  [2280] = {x=-3.091, y=2.427, z=22, rx=180, rz=-141.855, shoulder=lefty, elbow=epositive, wrist=wpositive, fatherId=fReference[0]}
  [2281] = {x=-1.854, y=1.456, z=22, rx=-180, rz=-141.854, shoulder=lefty, elbow=epositive, wrist=wpositive, fatherId=fReference[0]}
  [2282] = {x=-0.617, y=0.484, z=22, rx=-180, rz=-141.854, shoulder=lefty, elbow=epositive, wrist=wpositive, fatherId=fReference[0]}
  [2283] = {x=0.62, y=-0.487, z=22, rx=-180, rz=-141.854, shoulder=lefty, elbow=epositive, wrist=wpositive, fatherId=fReference[0]}
  [2284] = {x=1.857, y=-1.459, z=22, rx=180, rz=-141.855, shoulder=lefty, elbow=epositive, wrist=wpositive, fatherId=fReference[0]}
  [2285] = {x=3.094, y=-2.43, z=22, rx=-180, rz=-141.856, shoulder=lefty, elbow=epositive, wrist=wpositive, fatherId=fReference[0]}
  [2286] = {x=4.331, y=-3.402, z=22, rx=180, rz=-141.857, shoulder=lefty, elbow=epositive, wrist=wpositive, fatherId=fReference[0]}
  [2287] = {x=5.568, y=-4.373, z=22, rx=180, rz=-141.859, shoulder=lefty, elbow=epositive, wrist=wpositive, fatherId=fReference[0]}
  [2288] = {x=6.805, y=-5.345, z=22, rx=180, rz=-141.862, shoulder=lefty, elbow=epositive, wrist=wpositive, fatherId=fReference[0]}
  [2289] = {x=8.043, y=-6.316, z=22, rx=-180, rz=-141.864, shoulder=lefty, elbow=epositive, wrist=wpositive, fatherId=fReference[0]}
  [2290] = {x=9.28, y=-7.287, z=22, rx=180, rz=-141.867, shoulder=lefty, elbow=epositive, wrist=wpositive, fatherId=fReference[0]}
  [2291] = {x=10.517, y=-8.259, z=22, rx=-180, rz=-141.871, shoulder=lefty, elbow=epositive, wrist=wpositive, fatherId=fReference[0]}
  [2292] = {x=11.754, y=-9.23, z=22, rx=180, rz=-141.875, shoulder=lefty, elbow=epositive, wrist=wpositive, fatherId=fReference[0]}
  [2293] = {x=12.992, y=-10.201, z=22, rx=-180, rz=-141.879, shoulder=lefty, elbow=epositive, wrist=wpositive, fatherId=fReference[0]}
  [2294] = {x=14.229, y=-11.172, z=22, rx=-180, rz=-141.884, shoulder=lefty, elbow=epositive, wrist=wpositive, fatherId=fReference[0]}
  [2295] = {x=15.467, y=-12.143, z=22, rx=-180, rz=-141.89, shoulder=lefty, elbow=epositive, wrist=wpositive, fatherId=fReference[0]}
  [2296] = {x=16.704, y=-13.113, z=22, rx=180, rz=-141.895, shoulder=lefty, elbow=epositive, wrist=wpositive, fatherId=fReference[0]}
  [2297] = {x=17.942, y=-14.084, z=22, rx=-180, rz=-141.901, shoulder=lefty, elbow=epositive, wrist=wpositive, fatherId=fReference[0]}
  [2298] = {x=19.179, y=-15.054, z=22, rx=-180, rz=-141.908, shoulder=lefty, elbow=epositive, wrist=wpositive, fatherId=fReference[0]}
  [2299] = {x=20.417, y=-16.025, z=22, rx=-180, rz=-141.915, shoulder=lefty, elbow=epositive, wrist=wpositive, fatherId=fReference[0]}
  [2300] = {x=21.655, y=-16.995, z=22, rx=-180, rz=-141.922, shoulder=lefty, elbow=epositive, wrist=wpositive, fatherId=fReference[0]}
  [2301] = {x=22.893, y=-17.965, z=22, rx=180, rz=-141.93, shoulder=lefty, elbow=epositive, wrist=wpositive, fatherId=fReference[0]}
  [2302] = {x=24.131, y=-18.934, z=22, rx=-180, rz=-141.938, shoulder=lefty, elbow=epositive, wrist=wpositive, fatherId=fReference[0]}
  [2303] = {x=25.369, y=-19.904, z=22, rx=-180, rz=-141.947, shoulder=lefty, elbow=epositive, wrist=wpositive, fatherId=fReference[0]}
  [2304] = {x=26.607, y=-20.873, z=22, rx=180, rz=-141.956, shoulder=lefty, elbow=epositive, wrist=wpositive, fatherId=fReference[0]}
  [2305] = {x=27.846, y=-21.842, z=22, rx=180, rz=-141.965, shoulder=lefty, elbow=epositive, wrist=wpositive, fatherId=fReference[0]}
  [2306] = {x=29.084, y=-22.811, z=22, rx=180, rz=-141.975, shoulder=lefty, elbow=epositive, wrist=wpositive, fatherId=fReference[0]}
  [2307] = {x=30.323, y=-23.779, z=22, rx=-180, rz=-141.986, shoulder=lefty, elbow=epositive, wrist=wpositive, fatherId=fReference[0]}
  [2308] = {x=31.561, y=-24.748, z=22, rx=-180, rz=-141.996, shoulder=lefty, elbow=epositive, wrist=wpositive, fatherId=fReference[0]}
  [2309] = {x=32.8, y=-25.716, z=22, rx=180, rz=-142.008, shoulder=lefty, elbow=epositive, wrist=wpositive, fatherId=fReference[0]}
  [2310] = {x=34.039, y=-26.683, z=22, rx=-180, rz=-142.019, shoulder=lefty, elbow=epositive, wrist=wpositive, fatherId=fReference[0]}
  [2311] = {x=35.278, y=-27.651, z=22, rx=-180, rz=-142.031, shoulder=lefty, elbow=epositive, wrist=wpositive, fatherId=fReference[0]}
  [2312] = {x=36.517, y=-28.618, z=22, rx=-180, rz=-142.044, shoulder=lefty, elbow=epositive, wrist=wpositive, fatherId=fReference[0]}
  [2313] = {x=37.757, y=-29.585, z=22, rx=180, rz=-142.057, shoulder=lefty, elbow=epositive, wrist=wpositive, fatherId=fReference[0]}
  [2314] = {x=38.996, y=-30.551, z=22, rx=-180, rz=-142.07, shoulder=lefty, elbow=epositive, wrist=wpositive, fatherId=fReference[0]}
  [2315] = {x=40.236, y=-31.517, z=22, rx=180, rz=-142.084, shoulder=lefty, elbow=epositive, wrist=wpositive, fatherId=fReference[0]}
  [2316] = {x=41.476, y=-32.483, z=22, rx=180, rz=-142.098, shoulder=lefty, elbow=epositive, wrist=wpositive, fatherId=fReference[0]}
  [2317] = {x=42.715, y=-33.448, z=22, rx=-180, rz=-142.113, shoulder=lefty, elbow=epositive, wrist=wpositive, fatherId=fReference[0]}
  [2318] = {x=43.956, y=-34.413, z=22, rx=180, rz=-142.128, shoulder=lefty, elbow=epositive, wrist=wpositive, fatherId=fReference[0]}
  [2319] = {x=45.196, y=-35.377, z=22, rx=180, rz=-142.143, shoulder=lefty, elbow=epositive, wrist=wpositive, fatherId=fReference[0]}
  [2320] = {x=46.436, y=-36.342, z=22, rx=180, rz=-142.159, shoulder=lefty, elbow=epositive, wrist=wpositive, fatherId=fReference[0]}
  [2321] = {x=47.677, y=-37.305, z=22, rx=-180, rz=-142.175, shoulder=lefty, elbow=epositive, wrist=wpositive, fatherId=fReference[0]}
  [2322] = {x=48.917, y=-38.269, z=22, rx=-180, rz=-142.192, shoulder=lefty, elbow=epositive, wrist=wpositive, fatherId=fReference[0]}
  [2323] = {x=50.158, y=-39.231, z=22, rx=180, rz=-142.209, shoulder=lefty, elbow=epositive, wrist=wpositive, fatherId=fReference[0]}
  [2324] = {x=51.399, y=-40.194, z=22, rx=-180, rz=-142.227, shoulder=lefty, elbow=epositive, wrist=wpositive, fatherId=fReference[0]}
  [2325] = {x=52.641, y=-41.156, z=22, rx=180, rz=-142.245, shoulder=lefty, elbow=epositive, wrist=wpositive, fatherId=fReference[0]}
  [2326] = {x=53.882, y=-42.117, z=22, rx=-180, rz=-142.263, shoulder=lefty, elbow=epositive, wrist=wpositive, fatherId=fReference[0]}
  [2327] = {x=55.124, y=-43.078, z=22, rx=-180, rz=-142.282, shoulder=lefty, elbow=epositive, wrist=wpositive, fatherId=fReference[0]}
  [2328] = {x=56.366, y=-44.038, z=22, rx=180, rz=-142.302, shoulder=lefty, elbow=epositive, wrist=wpositive, fatherId=fReference[0]}
  [2329] = {x=57.608, y=-44.998, z=22, rx=-180, rz=-142.321, shoulder=lefty, elbow=epositive, wrist=wpositive, fatherId=fReference[0]}
  [2330] = {x=58.85, y=-45.958, z=22, rx=-180, rz=-142.342, shoulder=lefty, elbow=epositive, wrist=wpositive, fatherId=fReference[0]}
  [2331] = {x=60.092, y=-46.916, z=22, rx=-180, rz=-142.362, shoulder=lefty, elbow=epositive, wrist=wpositive, fatherId=fReference[0]}
  [2332] = {x=61.335, y=-47.875, z=22, rx=180, rz=-142.383, shoulder=lefty, elbow=epositive, wrist=wpositive, fatherId=fReference[0]}
  [2333] = {x=62.578, y=-48.832, z=22, rx=-180, rz=-142.405, shoulder=lefty, elbow=epositive, wrist=wpositive, fatherId=fReference[0]}
  [2334] = {x=63.821, y=-49.79, z=22, rx=-180, rz=-142.427, shoulder=lefty, elbow=epositive, wrist=wpositive, fatherId=fReference[0]}
  [2335] = {x=65.064, y=-50.746, z=22, rx=-180, rz=-142.449, shoulder=lefty, elbow=epositive, wrist=wpositive, fatherId=fReference[0]}
  [2336] = {x=66.308, y=-51.702, z=22, rx=-180, rz=-142.472, shoulder=lefty, elbow=epositive, wrist=wpositive, fatherId=fReference[0]}
  [2337] = {x=67.551, y=-52.657, z=22, rx=180, rz=-142.496, shoulder=lefty, elbow=epositive, wrist=wpositive, fatherId=fReference[0]}
  [2338] = {x=68.795, y=-53.612, z=22, rx=180, rz=-142.519, shoulder=lefty, elbow=epositive, wrist=wpositive, fatherId=fReference[0]}
  [2339] = {x=70.04, y=-54.566, z=22, rx=-180, rz=-142.543, shoulder=lefty, elbow=epositive, wrist=wpositive, fatherId=fReference[0]}
  [2340] = {x=71.284, y=-55.519, z=22, rx=-180, rz=-142.568, shoulder=lefty, elbow=epositive, wrist=wpositive, fatherId=fReference[0]}
  [2341] = {x=72.529, y=-56.472, z=22, rx=180, rz=-142.593, shoulder=lefty, elbow=epositive, wrist=wpositive, fatherId=fReference[0]}
  [2342] = {x=73.774, y=-57.424, z=22, rx=-180, rz=-142.619, shoulder=lefty, elbow=epositive, wrist=wpositive, fatherId=fReference[0]}
  [2343] = {x=75.019, y=-58.376, z=22, rx=180, rz=-142.645, shoulder=lefty, elbow=epositive, wrist=wpositive, fatherId=fReference[0]}
  [2344] = {x=76.264, y=-59.326, z=22, rx=-180, rz=-142.671, shoulder=lefty, elbow=epositive, wrist=wpositive, fatherId=fReference[0]}
  [2345] = {x=77.51, y=-60.276, z=22, rx=-180, rz=-142.698, shoulder=lefty, elbow=epositive, wrist=wpositive, fatherId=fReference[0]}
  [2346] = {x=78.756, y=-61.226, z=22, rx=-180, rz=-142.725, shoulder=lefty, elbow=epositive, wrist=wpositive, fatherId=fReference[0]}
  [2347] = {x=80.002, y=-62.174, z=22, rx=180, rz=-142.753, shoulder=lefty, elbow=epositive, wrist=wpositive, fatherId=fReference[0]}
  [2348] = {x=81.249, y=-63.122, z=22, rx=180, rz=-142.781, shoulder=lefty, elbow=epositive, wrist=wpositive, fatherId=fReference[0]}
  [2349] = {x=82.496, y=-64.069, z=22, rx=180, rz=-142.81, shoulder=lefty, elbow=epositive, wrist=wpositive, fatherId=fReference[0]}
  [2350] = {x=83.743, y=-65.015, z=22, rx=180, rz=-142.839, shoulder=lefty, elbow=epositive, wrist=wpositive, fatherId=fReference[0]}
  [2351] = {x=84.99, y=-65.961, z=22, rx=-180, rz=-142.868, shoulder=lefty, elbow=epositive, wrist=wpositive, fatherId=fReference[0]}
  [2352] = {x=86.238, y=-66.905, z=22, rx=-180, rz=-142.898, shoulder=lefty, elbow=epositive, wrist=wpositive, fatherId=fReference[0]}
  [2353] = {x=87.486, y=-67.849, z=22, rx=-180, rz=-142.929, shoulder=lefty, elbow=epositive, wrist=wpositive, fatherId=fReference[0]}
  [2354] = {x=88.734, y=-68.792, z=22, rx=-180, rz=-142.96, shoulder=lefty, elbow=epositive, wrist=wpositive, fatherId=fReference[0]}
  [2355] = {x=89.982, y=-69.734, z=22, rx=-180, rz=-142.991, shoulder=lefty, elbow=epositive, wrist=wpositive, fatherId=fReference[0]}
  [2356] = {x=91.231, y=-70.676, z=22, rx=-180, rz=-143.023, shoulder=lefty, elbow=epositive, wrist=wpositive, fatherId=fReference[0]}
  [2357] = {x=92.48, y=-71.616, z=22, rx=180, rz=-143.055, shoulder=lefty, elbow=epositive, wrist=wpositive, fatherId=fReference[0]}
  [2358] = {x=93.73, y=-72.556, z=22, rx=-180, rz=-143.088, shoulder=lefty, elbow=epositive, wrist=wpositive, fatherId=fReference[0]}
  [2359] = {x=94.979, y=-73.495, z=22, rx=-180, rz=-143.121, shoulder=lefty, elbow=epositive, wrist=wpositive, fatherId=fReference[0]}
  [2360] = {x=96.23, y=-74.432, z=22, rx=-180, rz=-143.155, shoulder=lefty, elbow=epositive, wrist=wpositive, fatherId=fReference[0]}
  [2361] = {x=97.48, y=-75.369, z=22, rx=180, rz=-143.189, shoulder=lefty, elbow=epositive, wrist=wpositive, fatherId=fReference[0]}
  [2362] = {x=98.731, y=-76.305, z=22, rx=-180, rz=-143.224, shoulder=lefty, elbow=epositive, wrist=wpositive, fatherId=fReference[0]}
  [2363] = {x=99.982, y=-77.24, z=22, rx=-180, rz=-143.259, shoulder=lefty, elbow=epositive, wrist=wpositive, fatherId=fReference[0]}
  [2364] = {x=101.233, y=-78.175, z=22, rx=-180, rz=-143.294, shoulder=lefty, elbow=epositive, wrist=wpositive, fatherId=fReference[0]}
  [2365] = {x=102.485, y=-79.108, z=22, rx=180, rz=-143.33, shoulder=lefty, elbow=epositive, wrist=wpositive, fatherId=fReference[0]}
  [2366] = {x=103.737, y=-80.04, z=22, rx=-180, rz=-143.367, shoulder=lefty, elbow=epositive, wrist=wpositive, fatherId=fReference[0]}
  [2367] = {x=104.989, y=-80.971, z=22, rx=-180, rz=-143.404, shoulder=lefty, elbow=epositive, wrist=wpositive, fatherId=fReference[0]}
  [2368] = {x=106.242, y=-81.901, z=22, rx=-180, rz=-143.441, shoulder=lefty, elbow=epositive, wrist=wpositive, fatherId=fReference[0]}
  [2369] = {x=107.495, y=-82.831, z=22, rx=-180, rz=-143.479, shoulder=lefty, elbow=epositive, wrist=wpositive, fatherId=fReference[0]}
  [2370] = {x=108.748, y=-83.759, z=22, rx=180, rz=-143.517, shoulder=lefty, elbow=epositive, wrist=wpositive, fatherId=fReference[0]}
  [2371] = {x=110.002, y=-84.686, z=22, rx=-180, rz=-143.556, shoulder=lefty, elbow=epositive, wrist=wpositive, fatherId=fReference[0]}
  [2372] = {x=111.256, y=-85.612, z=22, rx=-180, rz=-143.596, shoulder=lefty, elbow=epositive, wrist=wpositive, fatherId=fReference[0]}
  [2373] = {x=112.511, y=-86.537, z=22, rx=-180, rz=-143.635, shoulder=lefty, elbow=epositive, wrist=wpositive, fatherId=fReference[0]}
  [2374] = {x=113.766, y=-87.461, z=22, rx=180, rz=-143.676, shoulder=lefty, elbow=epositive, wrist=wpositive, fatherId=fReference[0]}
  [2375] = {x=115.021, y=-88.384, z=22, rx=180, rz=-143.716, shoulder=lefty, elbow=epositive, wrist=wpositive, fatherId=fReference[0]}
  [2376] = {x=116.277, y=-89.306, z=22, rx=-180, rz=-143.758, shoulder=lefty, elbow=epositive, wrist=wpositive, fatherId=fReference[0]}
  [2377] = {x=117.533, y=-90.227, z=22, rx=-180, rz=-143.799, shoulder=lefty, elbow=epositive, wrist=wpositive, fatherId=fReference[0]}
  [2378] = {x=118.789, y=-91.146, z=22, rx=-180, rz=-143.842, shoulder=lefty, elbow=epositive, wrist=wpositive, fatherId=fReference[0]}
  [2379] = {x=120.046, y=-92.065, z=22, rx=-180, rz=-143.884, shoulder=lefty, elbow=epositive, wrist=wpositive, fatherId=fReference[0]}
  [2380] = {x=121.304, y=-92.982, z=22, rx=-180, rz=-143.927, shoulder=lefty, elbow=epositive, wrist=wpositive, fatherId=fReference[0]}
  [2381] = {x=122.561, y=-93.898, z=22, rx=180, rz=-143.971, shoulder=lefty, elbow=epositive, wrist=wpositive, fatherId=fReference[0]}
  [2382] = {x=123.819, y=-94.813, z=22, rx=-180, rz=-144.015, shoulder=lefty, elbow=epositive, wrist=wpositive, fatherId=fReference[0]}
  [2383] = {x=125.078, y=-95.727, z=22, rx=180, rz=-144.06, shoulder=lefty, elbow=epositive, wrist=wpositive, fatherId=fReference[0]}
  [2384] = {x=126.337, y=-96.64, z=22, rx=-180, rz=-144.105, shoulder=lefty, elbow=epositive, wrist=wpositive, fatherId=fReference[0]}
  [2385] = {x=127.596, y=-97.551, z=22, rx=-180, rz=-144.151, shoulder=lefty, elbow=epositive, wrist=wpositive, fatherId=fReference[0]}
  [2386] = {x=128.856, y=-98.461, z=22, rx=-180, rz=-144.197, shoulder=lefty, elbow=epositive, wrist=wpositive, fatherId=fReference[0]}
  [2387] = {x=130.116, y=-99.37, z=22, rx=180, rz=-144.243, shoulder=lefty, elbow=epositive, wrist=wpositive, fatherId=fReference[0]}
  [2388] = {x=131.376, y=-100.278, z=22, rx=-180, rz=-144.291, shoulder=lefty, elbow=epositive, wrist=wpositive, fatherId=fReference[0]}
  [2389] = {x=132.637, y=-101.185, z=22, rx=180, rz=-144.338, shoulder=lefty, elbow=epositive, wrist=wpositive, fatherId=fReference[0]}
  [2390] = {x=133.899, y=-102.09, z=22, rx=-180, rz=-144.386, shoulder=lefty, elbow=epositive, wrist=wpositive, fatherId=fReference[0]}
  [2391] = {x=135.161, y=-102.994, z=22, rx=-180, rz=-144.435, shoulder=lefty, elbow=epositive, wrist=wpositive, fatherId=fReference[0]}
  [2392] = {x=136.423, y=-103.896, z=22, rx=180, rz=-144.484, shoulder=lefty, elbow=epositive, wrist=wpositive, fatherId=fReference[0]}
  [2393] = {x=137.686, y=-104.798, z=22, rx=180, rz=-144.534, shoulder=lefty, elbow=epositive, wrist=wpositive, fatherId=fReference[0]}
  [2394] = {x=138.949, y=-105.698, z=22, rx=180, rz=-144.584, shoulder=lefty, elbow=epositive, wrist=wpositive, fatherId=fReference[0]}
  [2395] = {x=140.213, y=-106.596, z=22, rx=180, rz=-144.634, shoulder=lefty, elbow=epositive, wrist=wpositive, fatherId=fReference[0]}
  [2396] = {x=141.477, y=-107.494, z=22, rx=-180, rz=-144.686, shoulder=lefty, elbow=epositive, wrist=wpositive, fatherId=fReference[0]}
  [2397] = {x=142.742, y=-108.389, z=22, rx=-180, rz=-144.737, shoulder=lefty, elbow=epositive, wrist=wpositive, fatherId=fReference[0]}
  [2398] = {x=144.007, y=-109.284, z=22, rx=-180, rz=-144.789, shoulder=lefty, elbow=epositive, wrist=wpositive, fatherId=fReference[0]}
  [2399] = {x=145.273, y=-110.177, z=22, rx=-180, rz=-144.842, shoulder=lefty, elbow=epositive, wrist=wpositive, fatherId=fReference[0]}
  [2400] = {x=146.539, y=-111.069, z=22, rx=-180, rz=-144.895, shoulder=lefty, elbow=epositive, wrist=wpositive, fatherId=fReference[0]}
  [2401] = {x=147.806, y=-111.959, z=22, rx=-180, rz=-144.949, shoulder=lefty, elbow=epositive, wrist=wpositive, fatherId=fReference[0]}
  [2402] = {x=149.073, y=-112.848, z=22, rx=-180, rz=-145.003, shoulder=lefty, elbow=epositive, wrist=wpositive, fatherId=fReference[0]}
  [2403] = {x=150.34, y=-113.736, z=22, rx=-180, rz=-145.058, shoulder=lefty, elbow=epositive, wrist=wpositive, fatherId=fReference[0]}
  [2404] = {x=151.608, y=-114.622, z=22, rx=-180, rz=-145.113, shoulder=lefty, elbow=epositive, wrist=wpositive, fatherId=fReference[0]}
  [2405] = {x=152.877, y=-115.506, z=22, rx=-180, rz=-145.169, shoulder=lefty, elbow=epositive, wrist=wpositive, fatherId=fReference[0]}
  [2406] = {x=154.146, y=-116.389, z=22, rx=180, rz=-145.225, shoulder=lefty, elbow=epositive, wrist=wpositive, fatherId=fReference[0]}
  [2407] = {x=155.416, y=-117.271, z=22, rx=180, rz=-145.282, shoulder=lefty, elbow=epositive, wrist=wpositive, fatherId=fReference[0]}
  [2408] = {x=156.686, y=-118.151, z=22, rx=-180, rz=-145.34, shoulder=lefty, elbow=epositive, wrist=wpositive, fatherId=fReference[0]}
  [2409] = {x=157.957, y=-119.03, z=22, rx=180, rz=-145.398, shoulder=lefty, elbow=epositive, wrist=wpositive, fatherId=fReference[0]}
  [2410] = {x=159.228, y=-119.907, z=22, rx=-180, rz=-145.456, shoulder=lefty, elbow=epositive, wrist=wpositive, fatherId=fReference[0]}
  [2411] = {x=160.5, y=-120.782, z=22, rx=-180, rz=-145.515, shoulder=lefty, elbow=epositive, wrist=wpositive, fatherId=fReference[0]}
  [2412] = {x=161.772, y=-121.656, z=22, rx=180, rz=-145.575, shoulder=lefty, elbow=epositive, wrist=wpositive, fatherId=fReference[0]}
  [2413] = {x=163.045, y=-122.529, z=22, rx=-180, rz=-145.635, shoulder=lefty, elbow=epositive, wrist=wpositive, fatherId=fReference[0]}
  [2414] = {x=164.319, y=-123.4, z=22, rx=-180, rz=-145.695, shoulder=lefty, elbow=epositive, wrist=wpositive, fatherId=fReference[0]}
  [2415] = {x=165.593, y=-124.269, z=22, rx=-180, rz=-145.756, shoulder=lefty, elbow=epositive, wrist=wpositive, fatherId=fReference[0]}
  [2416] = {x=166.867, y=-125.136, z=22, rx=-180, rz=-145.818, shoulder=lefty, elbow=epositive, wrist=wpositive, fatherId=fReference[0]}
  [2417] = {x=168.142, y=-126.002, z=22, rx=-180, rz=-145.88, shoulder=lefty, elbow=epositive, wrist=wpositive, fatherId=fReference[0]}
  [2418] = {x=169.418, y=-126.867, z=22, rx=-180, rz=-145.943, shoulder=lefty, elbow=epositive, wrist=wpositive, fatherId=fReference[0]}
  [2419] = {x=170.695, y=-127.73, z=22, rx=180, rz=-146.006, shoulder=lefty, elbow=epositive, wrist=wpositive, fatherId=fReference[0]}
  [2420] = {x=171.971, y=-128.591, z=22, rx=180, rz=-146.07, shoulder=lefty, elbow=epositive, wrist=wpositive, fatherId=fReference[0]}
  [2421] = {x=173.249, y=-129.45, z=22, rx=-180, rz=-146.135, shoulder=lefty, elbow=epositive, wrist=wpositive, fatherId=fReference[0]}
  [2422] = {x=174.527, y=-130.308, z=22, rx=180, rz=-146.2, shoulder=lefty, elbow=epositive, wrist=wpositive, fatherId=fReference[0]}
  [2423] = {x=175.806, y=-131.164, z=22, rx=-180, rz=-146.265, shoulder=lefty, elbow=epositive, wrist=wpositive, fatherId=fReference[0]}
  [2424] = {x=177.085, y=-132.018, z=22, rx=180, rz=-146.331, shoulder=lefty, elbow=epositive, wrist=wpositive, fatherId=fReference[0]}
  [2425] = {x=178.365, y=-132.871, z=22, rx=-180, rz=-146.398, shoulder=lefty, elbow=epositive, wrist=wpositive, fatherId=fReference[0]}
  [2426] = {x=179.645, y=-133.721, z=22, rx=-180, rz=-146.465, shoulder=lefty, elbow=epositive, wrist=wpositive, fatherId=fReference[0]}
  [2427] = {x=180.927, y=-134.571, z=22, rx=180, rz=-146.533, shoulder=lefty, elbow=epositive, wrist=wpositive, fatherId=fReference[0]}
  [2428] = {x=182.208, y=-135.418, z=22, rx=-180, rz=-146.601, shoulder=lefty, elbow=epositive, wrist=wpositive, fatherId=fReference[0]}
  [2429] = {x=183.491, y=-136.263, z=22, rx=-180, rz=-146.67, shoulder=lefty, elbow=epositive, wrist=wpositive, fatherId=fReference[0]}
  [2430] = {x=184.774, y=-137.107, z=22, rx=180, rz=-146.74, shoulder=lefty, elbow=epositive, wrist=wpositive, fatherId=fReference[0]}
  [2431] = {x=186.057, y=-137.949, z=22, rx=-180, rz=-146.81, shoulder=lefty, elbow=epositive, wrist=wpositive, fatherId=fReference[0]}
  [2432] = {x=187.341, y=-138.789, z=22, rx=180, rz=-146.881, shoulder=lefty, elbow=epositive, wrist=wpositive, fatherId=fReference[0]}
  [2433] = {x=188.626, y=-139.627, z=22, rx=-180, rz=-146.952, shoulder=lefty, elbow=epositive, wrist=wpositive, fatherId=fReference[0]}
  [2434] = {x=189.912, y=-140.464, z=22, rx=-180, rz=-147.024, shoulder=lefty, elbow=epositive, wrist=wpositive, fatherId=fReference[0]}
  [2435] = {x=191.198, y=-141.298, z=22, rx=-180, rz=-147.096, shoulder=lefty, elbow=epositive, wrist=wpositive, fatherId=fReference[0]}
  [2436] = {x=192.485, y=-142.131, z=22, rx=-180, rz=-147.169, shoulder=lefty, elbow=epositive, wrist=wpositive, fatherId=fReference[0]}
  [2437] = {x=193.772, y=-142.961, z=22, rx=-180, rz=-147.243, shoulder=lefty, elbow=epositive, wrist=wpositive, fatherId=fReference[0]}
  [2438] = {x=195.06, y=-143.79, z=22, rx=-180, rz=-147.317, shoulder=lefty, elbow=epositive, wrist=wpositive, fatherId=fReference[0]}
  [2439] = {x=196.349, y=-144.617, z=22, rx=-180, rz=-147.392, shoulder=lefty, elbow=epositive, wrist=wpositive, fatherId=fReference[0]}
  [2440] = {x=197.639, y=-145.442, z=22, rx=-180, rz=-147.467, shoulder=lefty, elbow=epositive, wrist=wpositive, fatherId=fReference[0]}
  [2441] = {x=198.929, y=-146.265, z=22, rx=-180, rz=-147.543, shoulder=lefty, elbow=epositive, wrist=wpositive, fatherId=fReference[0]}
  [2442] = {x=200.219, y=-147.086, z=22, rx=180, rz=-147.619, shoulder=lefty, elbow=epositive, wrist=wpositive, fatherId=fReference[0]}
  [2443] = {x=201.511, y=-147.905, z=22, rx=-180, rz=-147.697, shoulder=lefty, elbow=epositive, wrist=wpositive, fatherId=fReference[0]}
  [2444] = {x=202.803, y=-148.722, z=22, rx=-180, rz=-147.774, shoulder=lefty, elbow=epositive, wrist=wpositive, fatherId=fReference[0]}
  [2445] = {x=204.096, y=-149.536, z=22, rx=-180, rz=-147.853, shoulder=lefty, elbow=epositive, wrist=wpositive, fatherId=fReference[0]}
  [2446] = {x=205.389, y=-150.349, z=22, rx=-180, rz=-147.931, shoulder=lefty, elbow=epositive, wrist=wpositive, fatherId=fReference[0]}
  [2447] = {x=206.683, y=-151.16, z=22, rx=180, rz=-148.011, shoulder=lefty, elbow=epositive, wrist=wpositive, fatherId=fReference[0]}
  [2448] = {x=207.978, y=-151.969, z=22, rx=-180, rz=-148.091, shoulder=lefty, elbow=epositive, wrist=wpositive, fatherId=fReference[0]}
  [2449] = {x=209.273, y=-152.775, z=22, rx=-180, rz=-148.172, shoulder=lefty, elbow=epositive, wrist=wpositive, fatherId=fReference[0]}
  [2450] = {x=210.569, y=-153.58, z=22, rx=-180, rz=-148.253, shoulder=lefty, elbow=epositive, wrist=wpositive, fatherId=fReference[0]}
  [2451] = {x=211.866, y=-154.382, z=22, rx=-180, rz=-148.335, shoulder=lefty, elbow=epositive, wrist=wpositive, fatherId=fReference[0]}
  [2452] = {x=213.164, y=-155.183, z=22, rx=-180, rz=-148.418, shoulder=lefty, elbow=epositive, wrist=wpositive, fatherId=fReference[0]}
  [2453] = {x=214.462, y=-155.981, z=22, rx=-180, rz=-148.501, shoulder=lefty, elbow=epositive, wrist=wpositive, fatherId=fReference[0]}
  [2454] = {x=215.761, y=-156.777, z=22, rx=180, rz=-148.585, shoulder=lefty, elbow=epositive, wrist=wpositive, fatherId=fReference[0]}
  [2455] = {x=217.06, y=-157.57, z=22, rx=-180, rz=-148.669, shoulder=lefty, elbow=epositive, wrist=wpositive, fatherId=fReference[0]}
  [2456] = {x=218.361, y=-158.362, z=22, rx=-180, rz=-148.754, shoulder=lefty, elbow=epositive, wrist=wpositive, fatherId=fReference[0]}
  [2457] = {x=219.662, y=-159.151, z=22, rx=-180, rz=-148.84, shoulder=lefty, elbow=epositive, wrist=wpositive, fatherId=fReference[0]}
  [2458] = {x=220.963, y=-159.938, z=22, rx=-180, rz=-148.926, shoulder=lefty, elbow=epositive, wrist=wpositive, fatherId=fReference[0]}
  [2459] = {x=222.266, y=-160.723, z=22, rx=-180, rz=-149.013, shoulder=lefty, elbow=epositive, wrist=wpositive, fatherId=fReference[0]}
  [2460] = {x=223.569, y=-161.506, z=22, rx=-180, rz=-149.101, shoulder=lefty, elbow=epositive, wrist=wpositive, fatherId=fReference[0]}
  [2461] = {x=224.872, y=-162.286, z=22, rx=180, rz=-149.189, shoulder=lefty, elbow=epositive, wrist=wpositive, fatherId=fReference[0]}
  [2462] = {x=226.177, y=-163.064, z=22, rx=180, rz=-149.278, shoulder=lefty, elbow=epositive, wrist=wpositive, fatherId=fReference[0]}
  [2463] = {x=227.482, y=-163.84, z=22, rx=-180, rz=-149.367, shoulder=lefty, elbow=epositive, wrist=wpositive, fatherId=fReference[0]}
  [2464] = {x=228.788, y=-164.613, z=22, rx=-180, rz=-149.458, shoulder=lefty, elbow=epositive, wrist=wpositive, fatherId=fReference[0]}
  [2465] = {x=230.095, y=-165.384, z=22, rx=180, rz=-149.548, shoulder=lefty, elbow=epositive, wrist=wpositive, fatherId=fReference[0]}
  [2466] = {x=231.402, y=-166.152, z=22, rx=-180, rz=-149.64, shoulder=lefty, elbow=epositive, wrist=wpositive, fatherId=fReference[0]}
  [2467] = {x=232.71, y=-166.919, z=22, rx=-180, rz=-149.732, shoulder=lefty, elbow=epositive, wrist=wpositive, fatherId=fReference[0]}
  [2468] = {x=234.019, y=-167.682, z=22, rx=-180, rz=-149.824, shoulder=lefty, elbow=epositive, wrist=wpositive, fatherId=fReference[0]}
  [2469] = {x=235.328, y=-168.444, z=22, rx=-180, rz=-149.918, shoulder=lefty, elbow=epositive, wrist=wpositive, fatherId=fReference[0]}
  [2470] = {x=236.638, y=-169.203, z=22, rx=180, rz=-150.012, shoulder=lefty, elbow=epositive, wrist=wpositive, fatherId=fReference[0]}
  [2471] = {x=237.949, y=-169.959, z=22, rx=180, rz=-150.106, shoulder=lefty, elbow=epositive, wrist=wpositive, fatherId=fReference[0]}
  [2472] = {x=239.261, y=-170.713, z=22, rx=-180, rz=-150.202, shoulder=lefty, elbow=epositive, wrist=wpositive, fatherId=fReference[0]}
  [2473] = {x=240.573, y=-171.465, z=22, rx=-180, rz=-150.298, shoulder=lefty, elbow=epositive, wrist=wpositive, fatherId=fReference[0]}
  [2474] = {x=241.886, y=-172.214, z=22, rx=180, rz=-150.394, shoulder=lefty, elbow=epositive, wrist=wpositive, fatherId=fReference[0]}
  [2475] = {x=243.2, y=-172.96, z=22, rx=-180, rz=-150.491, shoulder=lefty, elbow=epositive, wrist=wpositive, fatherId=fReference[0]}
  [2476] = {x=244.514, y=-173.704, z=22, rx=-180, rz=-150.589, shoulder=lefty, elbow=epositive, wrist=wpositive, fatherId=fReference[0]}
  [2477] = {x=245.83, y=-174.446, z=22, rx=180, rz=-150.688, shoulder=lefty, elbow=epositive, wrist=wpositive, fatherId=fReference[0]}
  [2478] = {x=247.146, y=-175.184, z=22, rx=180, rz=-150.787, shoulder=lefty, elbow=epositive, wrist=wpositive, fatherId=fReference[0]}
  [2479] = {x=248.462, y=-175.921, z=22, rx=-180, rz=-150.887, shoulder=lefty, elbow=epositive, wrist=wpositive, fatherId=fReference[0]}
  [2480] = {x=249.78, y=-176.654, z=22, rx=-180, rz=-150.988, shoulder=lefty, elbow=epositive, wrist=wpositive, fatherId=fReference[0]}
  [2481] = {x=251.098, y=-177.385, z=22, rx=180, rz=-151.089, shoulder=lefty, elbow=epositive, wrist=wpositive, fatherId=fReference[0]}
  [2482] = {x=252.417, y=-178.114, z=22, rx=-180, rz=-151.191, shoulder=lefty, elbow=epositive, wrist=wpositive, fatherId=fReference[0]}
  [2483] = {x=253.736, y=-178.839, z=22, rx=180, rz=-151.293, shoulder=lefty, elbow=epositive, wrist=wpositive, fatherId=fReference[0]}
  [2484] = {x=255.056, y=-179.562, z=22, rx=-180, rz=-151.397, shoulder=lefty, elbow=epositive, wrist=wpositive, fatherId=fReference[0]}
  [2485] = {x=256.378, y=-180.283, z=22, rx=-180, rz=-151.501, shoulder=lefty, elbow=epositive, wrist=wpositive, fatherId=fReference[0]}
  [2486] = {x=257.699, y=-181, z=22, rx=-180, rz=-151.605, shoulder=lefty, elbow=epositive, wrist=wpositive, fatherId=fReference[0]}
  [2487] = {x=259.022, y=-181.715, z=22, rx=-180, rz=-151.711, shoulder=lefty, elbow=epositive, wrist=wpositive, fatherId=fReference[0]}
  [2488] = {x=260.345, y=-182.427, z=22, rx=-180, rz=-151.817, shoulder=lefty, elbow=epositive, wrist=wpositive, fatherId=fReference[0]}
  [2489] = {x=261.669, y=-183.137, z=22, rx=-180, rz=-151.923, shoulder=lefty, elbow=epositive, wrist=wpositive, fatherId=fReference[0]}
  [2490] = {x=262.994, y=-183.843, z=22, rx=-180, rz=-152.031, shoulder=lefty, elbow=epositive, wrist=wpositive, fatherId=fReference[0]}
  [2491] = {x=264.319, y=-184.547, z=22, rx=-180, rz=-152.139, shoulder=lefty, elbow=epositive, wrist=wpositive, fatherId=fReference[0]}
  [2492] = {x=265.645, y=-185.248, z=22, rx=-180, rz=-152.247, shoulder=lefty, elbow=epositive, wrist=wpositive, fatherId=fReference[0]}
  [2493] = {x=266.972, y=-185.946, z=22, rx=-180, rz=-152.357, shoulder=lefty, elbow=epositive, wrist=wpositive, fatherId=fReference[0]}
  [2494] = {x=268.3, y=-186.642, z=22, rx=-180, rz=-152.467, shoulder=lefty, elbow=epositive, wrist=wpositive, fatherId=fReference[0]}
  [2495] = {x=269.628, y=-187.334, z=22, rx=-180, rz=-152.578, shoulder=lefty, elbow=epositive, wrist=wpositive, fatherId=fReference[0]}
  [2496] = {x=270.957, y=-188.024, z=22, rx=180, rz=-152.689, shoulder=lefty, elbow=epositive, wrist=wpositive, fatherId=fReference[0]}
  [2497] = {x=272.287, y=-188.711, z=22, rx=180, rz=-152.801, shoulder=lefty, elbow=epositive, wrist=wpositive, fatherId=fReference[0]}
  [2498] = {x=273.617, y=-189.394, z=22, rx=180, rz=-152.914, shoulder=lefty, elbow=epositive, wrist=wpositive, fatherId=fReference[0]}
  [2499] = {x=274.948, y=-190.075, z=22, rx=-180, rz=-153.028, shoulder=lefty, elbow=epositive, wrist=wpositive, fatherId=fReference[0]}
  [2500] = {x=276.28, y=-190.753, z=22, rx=180, rz=-153.142, shoulder=lefty, elbow=epositive, wrist=wpositive, fatherId=fReference[0]}
  [2501] = {x=277.613, y=-191.428, z=22, rx=180, rz=-153.257, shoulder=lefty, elbow=epositive, wrist=wpositive, fatherId=fReference[0]}
  [2502] = {x=278.947, y=-192.1, z=22, rx=180, rz=-153.372, shoulder=lefty, elbow=epositive, wrist=wpositive, fatherId=fReference[0]}
  [2503] = {x=280.281, y=-192.769, z=22, rx=-180, rz=-153.489, shoulder=lefty, elbow=epositive, wrist=wpositive, fatherId=fReference[0]}
  [2504] = {x=281.616, y=-193.435, z=22, rx=-180, rz=-153.606, shoulder=lefty, elbow=epositive, wrist=wpositive, fatherId=fReference[0]}
  [2505] = {x=282.951, y=-194.097, z=22, rx=180, rz=-153.724, shoulder=lefty, elbow=epositive, wrist=wpositive, fatherId=fReference[0]}
  [2506] = {x=284.288, y=-194.757, z=22, rx=-180, rz=-153.842, shoulder=lefty, elbow=epositive, wrist=wpositive, fatherId=fReference[0]}
  [2507] = {x=285.625, y=-195.414, z=22, rx=-180, rz=-153.961, shoulder=lefty, elbow=epositive, wrist=wpositive, fatherId=fReference[0]}
  [2508] = {x=286.963, y=-196.068, z=22, rx=-180, rz=-154.081, shoulder=lefty, elbow=epositive, wrist=wpositive, fatherId=fReference[0]}
  [2509] = {x=288.301, y=-196.718, z=22, rx=-180, rz=-154.202, shoulder=lefty, elbow=epositive, wrist=wpositive, fatherId=fReference[0]}
  [2510] = {x=289.64, y=-197.365, z=22, rx=180, rz=-154.323, shoulder=lefty, elbow=epositive, wrist=wpositive, fatherId=fReference[0]}
  [2511] = {x=290.98, y=-198.01, z=22, rx=180, rz=-154.445, shoulder=lefty, elbow=epositive, wrist=wpositive, fatherId=fReference[0]}
  [2512] = {x=292.321, y=-198.651, z=22, rx=180, rz=-154.568, shoulder=lefty, elbow=epositive, wrist=wpositive, fatherId=fReference[0]}
  [2513] = {x=293.663, y=-199.289, z=22, rx=-180, rz=-154.691, shoulder=lefty, elbow=epositive, wrist=wpositive, fatherId=fReference[0]}
  [2514] = {x=295.005, y=-199.923, z=22, rx=-180, rz=-154.815, shoulder=lefty, elbow=epositive, wrist=wpositive, fatherId=fReference[0]}
  [2515] = {x=296.348, y=-200.555, z=22, rx=-180, rz=-154.94, shoulder=lefty, elbow=epositive, wrist=wpositive, fatherId=fReference[0]}
  [2516] = {x=297.691, y=-201.183, z=22, rx=-180, rz=-155.066, shoulder=lefty, elbow=epositive, wrist=wpositive, fatherId=fReference[0]}
  [2517] = {x=299.036, y=-201.808, z=22, rx=-180, rz=-155.192, shoulder=lefty, elbow=epositive, wrist=wpositive, fatherId=fReference[0]}
  [2518] = {x=300.381, y=-202.43, z=22, rx=-180, rz=-155.319, shoulder=lefty, elbow=epositive, wrist=wpositive, fatherId=fReference[0]}
  [2519] = {x=301.727, y=-203.048, z=22, rx=-180, rz=-155.447, shoulder=lefty, elbow=epositive, wrist=wpositive, fatherId=fReference[0]}
  [2520] = {x=303.073, y=-203.663, z=22, rx=180, rz=-155.575, shoulder=lefty, elbow=epositive, wrist=wpositive, fatherId=fReference[0]}
  [2521] = {x=304.421, y=-204.275, z=22, rx=-180, rz=-155.705, shoulder=lefty, elbow=epositive, wrist=wpositive, fatherId=fReference[0]}
  [2522] = {x=305.769, y=-204.884, z=22, rx=180, rz=-155.835, shoulder=lefty, elbow=epositive, wrist=wpositive, fatherId=fReference[0]}
  [2523] = {x=307.117, y=-205.489, z=22, rx=-180, rz=-155.965, shoulder=lefty, elbow=epositive, wrist=wpositive, fatherId=fReference[0]}
  [2524] = {x=308.467, y=-206.091, z=22, rx=180, rz=-156.097, shoulder=lefty, elbow=epositive, wrist=wpositive, fatherId=fReference[0]}
  [2525] = {x=309.817, y=-206.689, z=22, rx=180, rz=-156.229, shoulder=lefty, elbow=epositive, wrist=wpositive, fatherId=fReference[0]}
  [2526] = {x=311.168, y=-207.284, z=22, rx=-180, rz=-156.361, shoulder=lefty, elbow=epositive, wrist=wpositive, fatherId=fReference[0]}
  [2527] = {x=312.519, y=-207.876, z=22, rx=180, rz=-156.495, shoulder=lefty, elbow=epositive, wrist=wpositive, fatherId=fReference[0]}
  [2528] = {x=313.872, y=-208.464, z=22, rx=180, rz=-156.629, shoulder=lefty, elbow=epositive, wrist=wpositive, fatherId=fReference[0]}
  [2529] = {x=315.225, y=-209.049, z=22, rx=-180, rz=-156.764, shoulder=lefty, elbow=epositive, wrist=wpositive, fatherId=fReference[0]}
  [2530] = {x=316.579, y=-209.63, z=22, rx=-180, rz=-156.9, shoulder=lefty, elbow=epositive, wrist=wpositive, fatherId=fReference[0]}
  [2531] = {x=317.933, y=-210.208, z=22, rx=180, rz=-157.036, shoulder=lefty, elbow=epositive, wrist=wpositive, fatherId=fReference[0]}
  [2532] = {x=319.288, y=-210.782, z=22, rx=180, rz=-157.173, shoulder=lefty, elbow=epositive, wrist=wpositive, fatherId=fReference[0]}
  [2533] = {x=320.644, y=-211.353, z=22, rx=-180, rz=-157.311, shoulder=lefty, elbow=epositive, wrist=wpositive, fatherId=fReference[0]}
  [2534] = {x=322.001, y=-211.92, z=22, rx=180, rz=-157.45, shoulder=lefty, elbow=epositive, wrist=wpositive, fatherId=fReference[0]}
  [2535] = {x=323.358, y=-212.483, z=22, rx=180, rz=-157.589, shoulder=lefty, elbow=epositive, wrist=wpositive, fatherId=fReference[0]}
  [2536] = {x=324.716, y=-213.044, z=22, rx=-180, rz=-157.729, shoulder=lefty, elbow=epositive, wrist=wpositive, fatherId=fReference[0]}
  [2537] = {x=326.075, y=-213.6, z=22, rx=180, rz=-157.87, shoulder=lefty, elbow=epositive, wrist=wpositive, fatherId=fReference[0]}
  [2538] = {x=327.435, y=-214.153, z=22, rx=-180, rz=-158.011, shoulder=lefty, elbow=epositive, wrist=wpositive, fatherId=fReference[0]}
  [2539] = {x=328.795, y=-214.702, z=22, rx=180, rz=-158.153, shoulder=lefty, elbow=epositive, wrist=wpositive, fatherId=fReference[0]}
  [2540] = {x=330.156, y=-215.248, z=22, rx=180, rz=-158.296, shoulder=lefty, elbow=epositive, wrist=wpositive, fatherId=fReference[0]}
  [2541] = {x=331.517, y=-215.79, z=22, rx=-180, rz=-158.44, shoulder=lefty, elbow=epositive, wrist=wpositive, fatherId=fReference[0]}
  [2542] = {x=332.88, y=-216.328, z=22, rx=-180, rz=-158.584, shoulder=lefty, elbow=epositive, wrist=wpositive, fatherId=fReference[0]}
  [2543] = {x=334.243, y=-216.863, z=22, rx=180, rz=-158.729, shoulder=lefty, elbow=epositive, wrist=wpositive, fatherId=fReference[0]}
  [2544] = {x=335.607, y=-217.394, z=22, rx=180, rz=-158.875, shoulder=lefty, elbow=epositive, wrist=wpositive, fatherId=fReference[0]}
  [2545] = {x=336.971, y=-217.921, z=22, rx=180, rz=-159.022, shoulder=lefty, elbow=epositive, wrist=wpositive, fatherId=fReference[0]}
  [2546] = {x=338.336, y=-218.444, z=22, rx=180, rz=-159.169, shoulder=lefty, elbow=epositive, wrist=wpositive, fatherId=fReference[0]}
  [2547] = {x=339.702, y=-218.964, z=22, rx=-180, rz=-159.317, shoulder=lefty, elbow=epositive, wrist=wpositive, fatherId=fReference[0]}
  [2548] = {x=341.069, y=-219.48, z=22, rx=-180, rz=-159.465, shoulder=lefty, elbow=epositive, wrist=wpositive, fatherId=fReference[0]}
  [2549] = {x=342.436, y=-219.992, z=22, rx=-180, rz=-159.615, shoulder=lefty, elbow=epositive, wrist=wpositive, fatherId=fReference[0]}
  [2550] = {x=343.804, y=-220.5, z=22, rx=180, rz=-159.765, shoulder=lefty, elbow=epositive, wrist=wpositive, fatherId=fReference[0]}
  [2551] = {x=345.173, y=-221.005, z=22, rx=180, rz=-159.916, shoulder=lefty, elbow=epositive, wrist=wpositive, fatherId=fReference[0]}
  [2552] = {x=346.542, y=-221.506, z=22, rx=-180, rz=-160.067, shoulder=lefty, elbow=epositive, wrist=wpositive, fatherId=fReference[0]}
  [2553] = {x=347.912, y=-222.002, z=22, rx=-180, rz=-160.219, shoulder=lefty, elbow=epositive, wrist=wpositive, fatherId=fReference[0]}
  [2554] = {x=349.283, y=-222.495, z=22, rx=-180, rz=-160.372, shoulder=lefty, elbow=epositive, wrist=wpositive, fatherId=fReference[0]}
  [2555] = {x=350.655, y=-222.985, z=22, rx=-180, rz=-160.526, shoulder=lefty, elbow=epositive, wrist=wpositive, fatherId=fReference[0]}
  [2556] = {x=352.027, y=-223.47, z=22, rx=180, rz=-160.68, shoulder=lefty, elbow=epositive, wrist=wpositive, fatherId=fReference[0]}
  [2557] = {x=353.4, y=-223.951, z=22, rx=180, rz=-160.835, shoulder=lefty, elbow=epositive, wrist=wpositive, fatherId=fReference[0]}
  [2558] = {x=354.773, y=-224.429, z=22, rx=-180, rz=-160.991, shoulder=lefty, elbow=epositive, wrist=wpositive, fatherId=fReference[0]}
  [2559] = {x=356.148, y=-224.902, z=22, rx=180, rz=-161.147, shoulder=lefty, elbow=epositive, wrist=wpositive, fatherId=fReference[0]}
  [2560] = {x=357.523, y=-225.371, z=22, rx=-180, rz=-161.304, shoulder=lefty, elbow=epositive, wrist=wpositive, fatherId=fReference[0]}
  [2561] = {x=358.898, y=-225.837, z=22, rx=-180, rz=-161.462, shoulder=lefty, elbow=epositive, wrist=wpositive, fatherId=fReference[0]}
  [2562] = {x=360.275, y=-226.298, z=22, rx=-180, rz=-161.621, shoulder=lefty, elbow=epositive, wrist=wpositive, fatherId=fReference[0]}
  [2563] = {x=361.652, y=-226.756, z=22, rx=180, rz=-161.78, shoulder=lefty, elbow=epositive, wrist=wpositive, fatherId=fReference[0]}
  [2564] = {x=363.029, y=-227.209, z=22, rx=180, rz=-161.94, shoulder=lefty, elbow=epositive, wrist=wpositive, fatherId=fReference[0]}
  [2565] = {x=364.407, y=-227.659, z=22, rx=-180, rz=-162.1, shoulder=lefty, elbow=epositive, wrist=wpositive, fatherId=fReference[0]}
  [2566] = {x=365.786, y=-228.104, z=22, rx=-180, rz=-162.262, shoulder=lefty, elbow=epositive, wrist=wpositive, fatherId=fReference[0]}
  [2567] = {x=367.166, y=-228.546, z=22, rx=-180, rz=-162.424, shoulder=lefty, elbow=epositive, wrist=wpositive, fatherId=fReference[0]}
  [2568] = {x=368.546, y=-228.983, z=22, rx=180, rz=-162.586, shoulder=lefty, elbow=epositive, wrist=wpositive, fatherId=fReference[0]}
  [2569] = {x=369.927, y=-229.416, z=22, rx=180, rz=-162.75, shoulder=lefty, elbow=epositive, wrist=wpositive, fatherId=fReference[0]}
  [2570] = {x=371.309, y=-229.845, z=22, rx=-180, rz=-162.913, shoulder=lefty, elbow=epositive, wrist=wpositive, fatherId=fReference[0]}
  [2571] = {x=372.691, y=-230.27, z=22, rx=180, rz=-163.078, shoulder=lefty, elbow=epositive, wrist=wpositive, fatherId=fReference[0]}
  [2572] = {x=374.074, y=-230.69, z=22, rx=-180, rz=-163.243, shoulder=lefty, elbow=epositive, wrist=wpositive, fatherId=fReference[0]}
  [2573] = {x=375.457, y=-231.107, z=22, rx=-180, rz=-163.409, shoulder=lefty, elbow=epositive, wrist=wpositive, fatherId=fReference[0]}
  [2574] = {x=376.841, y=-231.519, z=22, rx=-180, rz=-163.576, shoulder=lefty, elbow=epositive, wrist=wpositive, fatherId=fReference[0]}
  [2575] = {x=378.226, y=-231.928, z=22, rx=180, rz=-163.743, shoulder=lefty, elbow=epositive, wrist=wpositive, fatherId=fReference[0]}
  [2576] = {x=379.611, y=-232.331, z=22, rx=-180, rz=-163.911, shoulder=lefty, elbow=epositive, wrist=wpositive, fatherId=fReference[0]}
  [2577] = {x=380.997, y=-232.731, z=22, rx=-180, rz=-164.08, shoulder=lefty, elbow=epositive, wrist=wpositive, fatherId=fReference[0]}
  [2578] = {x=382.384, y=-233.127, z=22, rx=-180, rz=-164.249, shoulder=lefty, elbow=epositive, wrist=wpositive, fatherId=fReference[0]}
  [2579] = {x=383.771, y=-233.518, z=22, rx=180, rz=-164.419, shoulder=lefty, elbow=epositive, wrist=wpositive, fatherId=fReference[0]}
  [2580] = {x=385.159, y=-233.905, z=22, rx=-180, rz=-164.589, shoulder=lefty, elbow=epositive, wrist=wpositive, fatherId=fReference[0]}
  [2581] = {x=386.547, y=-234.288, z=22, rx=-180, rz=-164.76, shoulder=lefty, elbow=epositive, wrist=wpositive, fatherId=fReference[0]}
  [2582] = {x=387.936, y=-234.666, z=22, rx=180, rz=-164.932, shoulder=lefty, elbow=epositive, wrist=wpositive, fatherId=fReference[0]}
  [2583] = {x=389.325, y=-235.04, z=22, rx=-180, rz=-165.105, shoulder=lefty, elbow=epositive, wrist=wpositive, fatherId=fReference[0]}
  [2584] = {x=390.715, y=-235.41, z=22, rx=-180, rz=-165.277, shoulder=lefty, elbow=epositive, wrist=wpositive, fatherId=fReference[0]}
  [2585] = {x=392.106, y=-235.775, z=22, rx=-180, rz=-165.451, shoulder=lefty, elbow=epositive, wrist=wpositive, fatherId=fReference[0]}
  [2586] = {x=393.497, y=-236.136, z=22, rx=-180, rz=-165.625, shoulder=lefty, elbow=epositive, wrist=wpositive, fatherId=fReference[0]}
  [2587] = {x=394.889, y=-236.493, z=22, rx=-180, rz=-165.8, shoulder=lefty, elbow=epositive, wrist=wpositive, fatherId=fReference[0]}
  [2588] = {x=396.281, y=-236.845, z=22, rx=-180, rz=-165.976, shoulder=lefty, elbow=epositive, wrist=wpositive, fatherId=fReference[0]}
  [2589] = {x=397.674, y=-237.193, z=22, rx=-180, rz=-166.152, shoulder=lefty, elbow=epositive, wrist=wpositive, fatherId=fReference[0]}
  [2590] = {x=399.068, y=-237.537, z=22, rx=-180, rz=-166.328, shoulder=lefty, elbow=epositive, wrist=wpositive, fatherId=fReference[0]}
  [2591] = {x=400.462, y=-237.876, z=22, rx=-180, rz=-166.505, shoulder=lefty, elbow=epositive, wrist=wpositive, fatherId=fReference[0]}
  [2592] = {x=401.856, y=-238.21, z=22, rx=-180, rz=-166.683, shoulder=lefty, elbow=epositive, wrist=wpositive, fatherId=fReference[0]}
  [2593] = {x=403.251, y=-238.541, z=22, rx=-180, rz=-166.861, shoulder=lefty, elbow=epositive, wrist=wpositive, fatherId=fReference[0]}
  [2594] = {x=404.647, y=-238.866, z=22, rx=-180, rz=-167.04, shoulder=lefty, elbow=epositive, wrist=wpositive, fatherId=fReference[0]}
  [2595] = {x=406.043, y=-239.188, z=22, rx=180, rz=-167.22, shoulder=lefty, elbow=epositive, wrist=wpositive, fatherId=fReference[0]}
  [2596] = {x=407.439, y=-239.505, z=22, rx=180, rz=-167.4, shoulder=lefty, elbow=epositive, wrist=wpositive, fatherId=fReference[0]}
  [2597] = {x=408.836, y=-239.817, z=22, rx=180, rz=-167.581, shoulder=lefty, elbow=epositive, wrist=wpositive, fatherId=fReference[0]}
  [2598] = {x=410.234, y=-240.125, z=22, rx=-180, rz=-167.762, shoulder=lefty, elbow=epositive, wrist=wpositive, fatherId=fReference[0]}
  [2599] = {x=411.632, y=-240.428, z=22, rx=180, rz=-167.943, shoulder=lefty, elbow=epositive, wrist=wpositive, fatherId=fReference[0]}
  [2600] = {x=413.031, y=-240.727, z=22, rx=-180, rz=-168.126, shoulder=lefty, elbow=epositive, wrist=wpositive, fatherId=fReference[0]}
  [2601] = {x=414.43, y=-241.021, z=22, rx=-180, rz=-168.308, shoulder=lefty, elbow=epositive, wrist=wpositive, fatherId=fReference[0]}
  [2602] = {x=415.829, y=-241.31, z=22, rx=180, rz=-168.492, shoulder=lefty, elbow=epositive, wrist=wpositive, fatherId=fReference[0]}
  [2603] = {x=417.229, y=-241.595, z=22, rx=180, rz=-168.675, shoulder=lefty, elbow=epositive, wrist=wpositive, fatherId=fReference[0]}
  [2604] = {x=418.63, y=-241.876, z=22, rx=180, rz=-168.86, shoulder=lefty, elbow=epositive, wrist=wpositive, fatherId=fReference[0]}
  [2605] = {x=420.031, y=-242.152, z=22, rx=180, rz=-169.045, shoulder=lefty, elbow=epositive, wrist=wpositive, fatherId=fReference[0]}
  [2606] = {x=421.432, y=-242.423, z=22, rx=-180, rz=-169.23, shoulder=lefty, elbow=epositive, wrist=wpositive, fatherId=fReference[0]}
  [2607] = {x=422.834, y=-242.69, z=22, rx=-180, rz=-169.416, shoulder=lefty, elbow=epositive, wrist=wpositive, fatherId=fReference[0]}
  [2608] = {x=424.236, y=-242.952, z=22, rx=-180, rz=-169.602, shoulder=lefty, elbow=epositive, wrist=wpositive, fatherId=fReference[0]}
  [2609] = {x=425.639, y=-243.209, z=22, rx=-180, rz=-169.789, shoulder=lefty, elbow=epositive, wrist=wpositive, fatherId=fReference[0]}
  [2610] = {x=427.042, y=-243.462, z=22, rx=-180, rz=-169.976, shoulder=lefty, elbow=epositive, wrist=wpositive, fatherId=fReference[0]}
  [2611] = {x=428.445, y=-243.71, z=22, rx=180, rz=-170.164, shoulder=lefty, elbow=epositive, wrist=wpositive, fatherId=fReference[0]}
  [2612] = {x=429.849, y=-243.953, z=22, rx=180, rz=-170.352, shoulder=lefty, elbow=epositive, wrist=wpositive, fatherId=fReference[0]}
  [2613] = {x=431.254, y=-244.192, z=22, rx=-180, rz=-170.54, shoulder=lefty, elbow=epositive, wrist=wpositive, fatherId=fReference[0]}
  [2614] = {x=432.658, y=-244.426, z=22, rx=-180, rz=-170.729, shoulder=lefty, elbow=epositive, wrist=wpositive, fatherId=fReference[0]}
  [2615] = {x=434.064, y=-244.655, z=22, rx=180, rz=-170.919, shoulder=lefty, elbow=epositive, wrist=wpositive, fatherId=fReference[0]}
  [2616] = {x=435.469, y=-244.88, z=22, rx=-180, rz=-171.109, shoulder=lefty, elbow=epositive, wrist=wpositive, fatherId=fReference[0]}
  [2617] = {x=436.875, y=-245.1, z=22, rx=-180, rz=-171.299, shoulder=lefty, elbow=epositive, wrist=wpositive, fatherId=fReference[0]}
  [2618] = {x=438.281, y=-245.315, z=22, rx=180, rz=-171.49, shoulder=lefty, elbow=epositive, wrist=wpositive, fatherId=fReference[0]}
  [2619] = {x=439.688, y=-245.526, z=22, rx=180, rz=-171.681, shoulder=lefty, elbow=epositive, wrist=wpositive, fatherId=fReference[0]}
  [2620] = {x=441.095, y=-245.731, z=22, rx=-180, rz=-171.873, shoulder=lefty, elbow=epositive, wrist=wpositive, fatherId=fReference[0]}
  [2621] = {x=442.502, y=-245.932, z=22, rx=-180, rz=-172.065, shoulder=lefty, elbow=epositive, wrist=wpositive, fatherId=fReference[0]}
  [2622] = {x=443.91, y=-246.129, z=22, rx=-180, rz=-172.257, shoulder=lefty, elbow=epositive, wrist=wpositive, fatherId=fReference[0]}
  [2623] = {x=445.318, y=-246.32, z=22, rx=-180, rz=-172.449, shoulder=lefty, elbow=epositive, wrist=wpositive, fatherId=fReference[0]}
  [2624] = {x=446.726, y=-246.507, z=22, rx=180, rz=-172.643, shoulder=lefty, elbow=epositive, wrist=wpositive, fatherId=fReference[0]}
  [2625] = {x=448.134, y=-246.689, z=22, rx=-180, rz=-172.836, shoulder=lefty, elbow=epositive, wrist=wpositive, fatherId=fReference[0]}
  [2626] = {x=449.543, y=-246.866, z=22, rx=-180, rz=-173.03, shoulder=lefty, elbow=epositive, wrist=wpositive, fatherId=fReference[0]}
  [2627] = {x=450.953, y=-247.038, z=22, rx=180, rz=-173.224, shoulder=lefty, elbow=epositive, wrist=wpositive, fatherId=fReference[0]}
  [2628] = {x=452.362, y=-247.205, z=22, rx=180, rz=-173.418, shoulder=lefty, elbow=epositive, wrist=wpositive, fatherId=fReference[0]}
  [2629] = {x=453.772, y=-247.368, z=22, rx=180, rz=-173.613, shoulder=lefty, elbow=epositive, wrist=wpositive, fatherId=fReference[0]}
  [2630] = {x=455.182, y=-247.526, z=22, rx=180, rz=-173.808, shoulder=lefty, elbow=epositive, wrist=wpositive, fatherId=fReference[0]}
  [2631] = {x=456.592, y=-247.679, z=22, rx=-180, rz=-174.003, shoulder=lefty, elbow=epositive, wrist=wpositive, fatherId=fReference[0]}
  [2632] = {x=458.003, y=-247.827, z=22, rx=180, rz=-174.199, shoulder=lefty, elbow=epositive, wrist=wpositive, fatherId=fReference[0]}
  [2633] = {x=459.414, y=-247.971, z=22, rx=-180, rz=-174.395, shoulder=lefty, elbow=epositive, wrist=wpositive, fatherId=fReference[0]}
  [2634] = {x=460.825, y=-248.109, z=22, rx=-180, rz=-174.591, shoulder=lefty, elbow=epositive, wrist=wpositive, fatherId=fReference[0]}
  [2635] = {x=462.236, y=-248.243, z=22, rx=-180, rz=-174.787, shoulder=lefty, elbow=epositive, wrist=wpositive, fatherId=fReference[0]}
  [2636] = {x=463.647, y=-248.371, z=22, rx=180, rz=-174.984, shoulder=lefty, elbow=epositive, wrist=wpositive, fatherId=fReference[0]}
  [2637] = {x=465.059, y=-248.495, z=22, rx=180, rz=-175.181, shoulder=lefty, elbow=epositive, wrist=wpositive, fatherId=fReference[0]}
  [2638] = {x=466.471, y=-248.614, z=22, rx=180, rz=-175.378, shoulder=lefty, elbow=epositive, wrist=wpositive, fatherId=fReference[0]}
  [2639] = {x=467.883, y=-248.729, z=22, rx=180, rz=-175.575, shoulder=lefty, elbow=epositive, wrist=wpositive, fatherId=fReference[0]}
  [2640] = {x=469.296, y=-248.838, z=22, rx=-180, rz=-175.773, shoulder=lefty, elbow=epositive, wrist=wpositive, fatherId=fReference[0]}
  [2641] = {x=470.708, y=-248.942, z=22, rx=-180, rz=-175.971, shoulder=lefty, elbow=epositive, wrist=wpositive, fatherId=fReference[0]}
  [2642] = {x=472.121, y=-249.042, z=22, rx=180, rz=-176.169, shoulder=lefty, elbow=epositive, wrist=wpositive, fatherId=fReference[0]}
  [2643] = {x=473.534, y=-249.136, z=22, rx=-180, rz=-176.367, shoulder=lefty, elbow=epositive, wrist=wpositive, fatherId=fReference[0]}
  [2644] = {x=474.947, y=-249.226, z=22, rx=-180, rz=-176.566, shoulder=lefty, elbow=epositive, wrist=wpositive, fatherId=fReference[0]}
  [2645] = {x=476.36, y=-249.311, z=22, rx=180, rz=-176.764, shoulder=lefty, elbow=epositive, wrist=wpositive, fatherId=fReference[0]}
  [2646] = {x=477.773, y=-249.391, z=22, rx=180, rz=-176.963, shoulder=lefty, elbow=epositive, wrist=wpositive, fatherId=fReference[0]}
  [2647] = {x=479.187, y=-249.466, z=22, rx=-180, rz=-177.162, shoulder=lefty, elbow=epositive, wrist=wpositive, fatherId=fReference[0]}
  [2648] = {x=480.6, y=-249.536, z=22, rx=-180, rz=-177.361, shoulder=lefty, elbow=epositive, wrist=wpositive, fatherId=fReference[0]}
  [2649] = {x=482.014, y=-249.601, z=22, rx=-180, rz=-177.56, shoulder=lefty, elbow=epositive, wrist=wpositive, fatherId=fReference[0]}
  [2650] = {x=483.428, y=-249.661, z=22, rx=-180, rz=-177.759, shoulder=lefty, elbow=epositive, wrist=wpositive, fatherId=fReference[0]}
  [2651] = {x=484.841, y=-249.717, z=22, rx=-180, rz=-177.959, shoulder=lefty, elbow=epositive, wrist=wpositive, fatherId=fReference[0]}
  [2652] = {x=486.255, y=-249.767, z=22, rx=-180, rz=-178.158, shoulder=lefty, elbow=epositive, wrist=wpositive, fatherId=fReference[0]}
  [2653] = {x=487.669, y=-249.812, z=22, rx=-180, rz=-178.358, shoulder=lefty, elbow=epositive, wrist=wpositive, fatherId=fReference[0]}
  [2654] = {x=489.084, y=-249.853, z=22, rx=-180, rz=-178.557, shoulder=lefty, elbow=epositive, wrist=wpositive, fatherId=fReference[0]}
  [2655] = {x=490.498, y=-249.889, z=22, rx=180, rz=-178.757, shoulder=lefty, elbow=epositive, wrist=wpositive, fatherId=fReference[0]}
  [2656] = {x=491.912, y=-249.919, z=22, rx=180, rz=-178.957, shoulder=lefty, elbow=epositive, wrist=wpositive, fatherId=fReference[0]}
  [2657] = {x=493.326, y=-249.945, z=22, rx=-180, rz=-179.157, shoulder=lefty, elbow=epositive, wrist=wpositive, fatherId=fReference[0]}
  [2658] = {x=494.741, y=-249.966, z=22, rx=-180, rz=-179.357, shoulder=lefty, elbow=epositive, wrist=wpositive, fatherId=fReference[0]}
  [2659] = {x=496.155, y=-249.982, z=22, rx=-180, rz=-179.557, shoulder=lefty, elbow=epositive, wrist=wpositive, fatherId=fReference[0]}
  [2660] = {x=497.569, y=-249.993, z=22, rx=-180, rz=-179.756, shoulder=lefty, elbow=epositive, wrist=wpositive, fatherId=fReference[0]}
  [2661] = {x=498.984, y=-249.999, z=22, rx=-180, rz=-179.956, shoulder=lefty, elbow=epositive, wrist=wpositive, fatherId=fReference[0]}
  [2662] = {x=500.398, y=-250, z=22, rx=-180, rz=179.844, shoulder=lefty, elbow=epositive, wrist=wpositive, fatherId=fReference[0]}
  [2663] = {x=501.812, y=-249.996, z=22, rx=180, rz=179.644, shoulder=lefty, elbow=epositive, wrist=wpositive, fatherId=fReference[0]}
  [2664] = {x=503.227, y=-249.987, z=22, rx=-180, rz=179.444, shoulder=lefty, elbow=epositive, wrist=wpositive, fatherId=fReference[0]}
  [2665] = {x=504.641, y=-249.973, z=22, rx=180, rz=179.244, shoulder=lefty, elbow=epositive, wrist=wpositive, fatherId=fReference[0]}
  [2666] = {x=506.055, y=-249.955, z=22, rx=-180, rz=179.044, shoulder=lefty, elbow=epositive, wrist=wpositive, fatherId=fReference[0]}
  [2667] = {x=507.47, y=-249.931, z=22, rx=-180, rz=178.844, shoulder=lefty, elbow=epositive, wrist=wpositive, fatherId=fReference[0]}
  [2668] = {x=508.884, y=-249.903, z=22, rx=-180, rz=178.645, shoulder=lefty, elbow=epositive, wrist=wpositive, fatherId=fReference[0]}
  [2669] = {x=510.298, y=-249.869, z=22, rx=-180, rz=178.445, shoulder=lefty, elbow=epositive, wrist=wpositive, fatherId=fReference[0]}
  [2670] = {x=511.712, y=-249.831, z=22, rx=180, rz=178.245, shoulder=lefty, elbow=epositive, wrist=wpositive, fatherId=fReference[0]}
  [2671] = {x=513.126, y=-249.787, z=22, rx=-180, rz=178.046, shoulder=lefty, elbow=epositive, wrist=wpositive, fatherId=fReference[0]}
  [2672] = {x=514.54, y=-249.739, z=22, rx=180, rz=177.846, shoulder=lefty, elbow=epositive, wrist=wpositive, fatherId=fReference[0]}
  [2673] = {x=515.954, y=-249.686, z=22, rx=180, rz=177.647, shoulder=lefty, elbow=epositive, wrist=wpositive, fatherId=fReference[0]}
  [2674] = {x=517.368, y=-249.628, z=22, rx=180, rz=177.448, shoulder=lefty, elbow=epositive, wrist=wpositive, fatherId=fReference[0]}
  [2675] = {x=518.782, y=-249.565, z=22, rx=180, rz=177.249, shoulder=lefty, elbow=epositive, wrist=wpositive, fatherId=fReference[0]}
  [2676] = {x=520.195, y=-249.497, z=22, rx=-180, rz=177.05, shoulder=lefty, elbow=epositive, wrist=wpositive, fatherId=fReference[0]}
  [2677] = {x=521.609, y=-249.424, z=22, rx=-180, rz=176.851, shoulder=lefty, elbow=epositive, wrist=wpositive, fatherId=fReference[0]}
  [2678] = {x=523.022, y=-249.346, z=22, rx=180, rz=176.652, shoulder=lefty, elbow=epositive, wrist=wpositive, fatherId=fReference[0]}
  [2679] = {x=524.435, y=-249.264, z=22, rx=-180, rz=176.454, shoulder=lefty, elbow=epositive, wrist=wpositive, fatherId=fReference[0]}
  [2680] = {x=525.848, y=-249.176, z=22, rx=-180, rz=176.256, shoulder=lefty, elbow=epositive, wrist=wpositive, fatherId=fReference[0]}
  [2681] = {x=527.261, y=-249.084, z=22, rx=180, rz=176.058, shoulder=lefty, elbow=epositive, wrist=wpositive, fatherId=fReference[0]}
  [2682] = {x=528.674, y=-248.986, z=22, rx=180, rz=175.86, shoulder=lefty, elbow=epositive, wrist=wpositive, fatherId=fReference[0]}
  [2683] = {x=530.086, y=-248.884, z=22, rx=180, rz=175.662, shoulder=lefty, elbow=epositive, wrist=wpositive, fatherId=fReference[0]}
  [2684] = {x=531.498, y=-248.777, z=22, rx=180, rz=175.465, shoulder=lefty, elbow=epositive, wrist=wpositive, fatherId=fReference[0]}
  [2685] = {x=532.911, y=-248.665, z=22, rx=180, rz=175.267, shoulder=lefty, elbow=epositive, wrist=wpositive, fatherId=fReference[0]}
  [2686] = {x=534.323, y=-248.548, z=22, rx=-180, rz=175.07, shoulder=lefty, elbow=epositive, wrist=wpositive, fatherId=fReference[0]}
  [2687] = {x=535.734, y=-248.426, z=22, rx=-180, rz=174.874, shoulder=lefty, elbow=epositive, wrist=wpositive, fatherId=fReference[0]}
  [2688] = {x=537.146, y=-248.3, z=22, rx=-180, rz=174.677, shoulder=lefty, elbow=epositive, wrist=wpositive, fatherId=fReference[0]}
  [2689] = {x=538.557, y=-248.168, z=22, rx=-180, rz=174.481, shoulder=lefty, elbow=epositive, wrist=wpositive, fatherId=fReference[0]}
  [2690] = {x=539.968, y=-248.032, z=22, rx=-180, rz=174.285, shoulder=lefty, elbow=epositive, wrist=wpositive, fatherId=fReference[0]}
  [2691] = {x=541.379, y=-247.891, z=22, rx=180, rz=174.089, shoulder=lefty, elbow=epositive, wrist=wpositive, fatherId=fReference[0]}
  [2692] = {x=542.79, y=-247.744, z=22, rx=-180, rz=173.894, shoulder=lefty, elbow=epositive, wrist=wpositive, fatherId=fReference[0]}
  [2693] = {x=544.2, y=-247.594, z=22, rx=-180, rz=173.698, shoulder=lefty, elbow=epositive, wrist=wpositive, fatherId=fReference[0]}
  [2694] = {x=545.61, y=-247.438, z=22, rx=180, rz=173.504, shoulder=lefty, elbow=epositive, wrist=wpositive, fatherId=fReference[0]}
  [2695] = {x=547.02, y=-247.277, z=22, rx=180, rz=173.309, shoulder=lefty, elbow=epositive, wrist=wpositive, fatherId=fReference[0]}
  [2696] = {x=548.43, y=-247.112, z=22, rx=180, rz=173.115, shoulder=lefty, elbow=epositive, wrist=wpositive, fatherId=fReference[0]}
  [2697] = {x=549.839, y=-246.942, z=22, rx=180, rz=172.921, shoulder=lefty, elbow=epositive, wrist=wpositive, fatherId=fReference[0]}
  [2698] = {x=551.248, y=-246.767, z=22, rx=-180, rz=172.727, shoulder=lefty, elbow=epositive, wrist=wpositive, fatherId=fReference[0]}
  [2699] = {x=552.657, y=-246.587, z=22, rx=180, rz=172.534, shoulder=lefty, elbow=epositive, wrist=wpositive, fatherId=fReference[0]}
  [2700] = {x=554.065, y=-246.402, z=22, rx=-180, rz=172.341, shoulder=lefty, elbow=epositive, wrist=wpositive, fatherId=fReference[0]}
  [2701] = {x=555.473, y=-246.213, z=22, rx=-180, rz=172.149, shoulder=lefty, elbow=epositive, wrist=wpositive, fatherId=fReference[0]}
  [2702] = {x=556.881, y=-246.019, z=22, rx=180, rz=171.957, shoulder=lefty, elbow=epositive, wrist=wpositive, fatherId=fReference[0]}
  [2703] = {x=558.289, y=-245.82, z=22, rx=-180, rz=171.765, shoulder=lefty, elbow=epositive, wrist=wpositive, fatherId=fReference[0]}
  [2704] = {x=559.696, y=-245.616, z=22, rx=180, rz=171.574, shoulder=lefty, elbow=epositive, wrist=wpositive, fatherId=fReference[0]}
  [2705] = {x=561.102, y=-245.408, z=22, rx=180, rz=171.383, shoulder=lefty, elbow=epositive, wrist=wpositive, fatherId=fReference[0]}
  [2706] = {x=562.509, y=-245.195, z=22, rx=-180, rz=171.192, shoulder=lefty, elbow=epositive, wrist=wpositive, fatherId=fReference[0]}
  [2707] = {x=563.915, y=-244.977, z=22, rx=180, rz=171.002, shoulder=lefty, elbow=epositive, wrist=wpositive, fatherId=fReference[0]}
  [2708] = {x=565.321, y=-244.755, z=22, rx=180, rz=170.813, shoulder=lefty, elbow=epositive, wrist=wpositive, fatherId=fReference[0]}
  [2709] = {x=566.726, y=-244.527, z=22, rx=-180, rz=170.623, shoulder=lefty, elbow=epositive, wrist=wpositive, fatherId=fReference[0]}
  [2710] = {x=568.131, y=-244.295, z=22, rx=-180, rz=170.435, shoulder=lefty, elbow=epositive, wrist=wpositive, fatherId=fReference[0]}
  [2711] = {x=569.535, y=-244.059, z=22, rx=-180, rz=170.246, shoulder=lefty, elbow=epositive, wrist=wpositive, fatherId=fReference[0]}
  [2712] = {x=570.939, y=-243.817, z=22, rx=180, rz=170.058, shoulder=lefty, elbow=epositive, wrist=wpositive, fatherId=fReference[0]}
  [2713] = {x=572.343, y=-243.571, z=22, rx=180, rz=169.871, shoulder=lefty, elbow=epositive, wrist=wpositive, fatherId=fReference[0]}
  [2714] = {x=573.746, y=-243.32, z=22, rx=180, rz=169.684, shoulder=lefty, elbow=epositive, wrist=wpositive, fatherId=fReference[0]}
  [2715] = {x=575.149, y=-243.065, z=22, rx=-180, rz=169.497, shoulder=lefty, elbow=epositive, wrist=wpositive, fatherId=fReference[0]}
  [2716] = {x=576.552, y=-242.805, z=22, rx=180, rz=169.311, shoulder=lefty, elbow=epositive, wrist=wpositive, fatherId=fReference[0]}
  [2717] = {x=577.954, y=-242.54, z=22, rx=-180, rz=169.126, shoulder=lefty, elbow=epositive, wrist=wpositive, fatherId=fReference[0]}
  [2718] = {x=579.355, y=-242.271, z=22, rx=-180, rz=168.941, shoulder=lefty, elbow=epositive, wrist=wpositive, fatherId=fReference[0]}
  [2719] = {x=580.757, y=-241.997, z=22, rx=-180, rz=168.756, shoulder=lefty, elbow=epositive, wrist=wpositive, fatherId=fReference[0]}
  [2720] = {x=582.157, y=-241.719, z=22, rx=180, rz=168.572, shoulder=lefty, elbow=epositive, wrist=wpositive, fatherId=fReference[0]}
  [2721] = {x=583.557, y=-241.436, z=22, rx=-180, rz=168.389, shoulder=lefty, elbow=epositive, wrist=wpositive, fatherId=fReference[0]}
  [2722] = {x=584.957, y=-241.148, z=22, rx=-180, rz=168.206, shoulder=lefty, elbow=epositive, wrist=wpositive, fatherId=fReference[0]}
  [2723] = {x=586.357, y=-240.856, z=22, rx=-180, rz=168.023, shoulder=lefty, elbow=epositive, wrist=wpositive, fatherId=fReference[0]}
  [2724] = {x=587.755, y=-240.559, z=22, rx=180, rz=167.841, shoulder=lefty, elbow=epositive, wrist=wpositive, fatherId=fReference[0]}
  [2725] = {x=589.154, y=-240.258, z=22, rx=180, rz=167.66, shoulder=lefty, elbow=epositive, wrist=wpositive, fatherId=fReference[0]}
  [2726] = {x=590.552, y=-239.952, z=22, rx=-180, rz=167.479, shoulder=lefty, elbow=epositive, wrist=wpositive, fatherId=fReference[0]}
  [2727] = {x=591.949, y=-239.642, z=22, rx=-180, rz=167.299, shoulder=lefty, elbow=epositive, wrist=wpositive, fatherId=fReference[0]}
  [2728] = {x=593.346, y=-239.327, z=22, rx=180, rz=167.119, shoulder=lefty, elbow=epositive, wrist=wpositive, fatherId=fReference[0]}
  [2729] = {x=594.742, y=-239.008, z=22, rx=180, rz=166.94, shoulder=lefty, elbow=epositive, wrist=wpositive, fatherId=fReference[0]}
  [2730] = {x=596.138, y=-238.684, z=22, rx=180, rz=166.761, shoulder=lefty, elbow=epositive, wrist=wpositive, fatherId=fReference[0]}
  [2731] = {x=597.533, y=-238.356, z=22, rx=180, rz=166.583, shoulder=lefty, elbow=epositive, wrist=wpositive, fatherId=fReference[0]}
  [2732] = {x=598.928, y=-238.023, z=22, rx=180, rz=166.405, shoulder=lefty, elbow=epositive, wrist=wpositive, fatherId=fReference[0]}
  [2733] = {x=600.322, y=-237.686, z=22, rx=180, rz=166.229, shoulder=lefty, elbow=epositive, wrist=wpositive, fatherId=fReference[0]}
  [2734] = {x=601.716, y=-237.344, z=22, rx=-180, rz=166.052, shoulder=lefty, elbow=epositive, wrist=wpositive, fatherId=fReference[0]}
  [2735] = {x=603.109, y=-236.998, z=22, rx=-180, rz=165.877, shoulder=lefty, elbow=epositive, wrist=wpositive, fatherId=fReference[0]}
  [2736] = {x=604.502, y=-236.648, z=22, rx=-180, rz=165.702, shoulder=lefty, elbow=epositive, wrist=wpositive, fatherId=fReference[0]}
  [2737] = {x=605.894, y=-236.293, z=22, rx=-180, rz=165.527, shoulder=lefty, elbow=epositive, wrist=wpositive, fatherId=fReference[0]}
  [2738] = {x=607.286, y=-235.934, z=22, rx=-180, rz=165.353, shoulder=lefty, elbow=epositive, wrist=wpositive, fatherId=fReference[0]}
  [2739] = {x=608.677, y=-235.57, z=22, rx=-180, rz=165.18, shoulder=lefty, elbow=epositive, wrist=wpositive, fatherId=fReference[0]}
  [2740] = {x=610.067, y=-235.202, z=22, rx=-180, rz=165.007, shoulder=lefty, elbow=epositive, wrist=wpositive, fatherId=fReference[0]}
  [2741] = {x=611.457, y=-234.83, z=22, rx=180, rz=164.835, shoulder=lefty, elbow=epositive, wrist=wpositive, fatherId=fReference[0]}
  [2742] = {x=612.846, y=-234.454, z=22, rx=-180, rz=164.664, shoulder=lefty, elbow=epositive, wrist=wpositive, fatherId=fReference[0]}
  [2743] = {x=614.235, y=-234.073, z=22, rx=180, rz=164.493, shoulder=lefty, elbow=epositive, wrist=wpositive, fatherId=fReference[0]}
  [2744] = {x=615.623, y=-233.688, z=22, rx=-180, rz=164.323, shoulder=lefty, elbow=epositive, wrist=wpositive, fatherId=fReference[0]}
  [2745] = {x=617.01, y=-233.298, z=22, rx=180, rz=164.153, shoulder=lefty, elbow=epositive, wrist=wpositive, fatherId=fReference[0]}
  [2746] = {x=618.397, y=-232.905, z=22, rx=-180, rz=163.985, shoulder=lefty, elbow=epositive, wrist=wpositive, fatherId=fReference[0]}
  [2747] = {x=619.783, y=-232.507, z=22, rx=-180, rz=163.816, shoulder=lefty, elbow=epositive, wrist=wpositive, fatherId=fReference[0]}
  [2748] = {x=621.169, y=-232.104, z=22, rx=-180, rz=163.649, shoulder=lefty, elbow=epositive, wrist=wpositive, fatherId=fReference[0]}
  [2749] = {x=622.554, y=-231.698, z=22, rx=180, rz=163.482, shoulder=lefty, elbow=epositive, wrist=wpositive, fatherId=fReference[0]}
  [2750] = {x=623.939, y=-231.288, z=22, rx=-180, rz=163.316, shoulder=lefty, elbow=epositive, wrist=wpositive, fatherId=fReference[0]}
  [2751] = {x=625.322, y=-230.873, z=22, rx=-180, rz=163.15, shoulder=lefty, elbow=epositive, wrist=wpositive, fatherId=fReference[0]}
  [2752] = {x=626.706, y=-230.454, z=22, rx=-180, rz=162.985, shoulder=lefty, elbow=epositive, wrist=wpositive, fatherId=fReference[0]}
  [2753] = {x=628.088, y=-230.031, z=22, rx=180, rz=162.821, shoulder=lefty, elbow=epositive, wrist=wpositive, fatherId=fReference[0]}
  [2754] = {x=629.47, y=-229.604, z=22, rx=180, rz=162.657, shoulder=lefty, elbow=epositive, wrist=wpositive, fatherId=fReference[0]}
  [2755] = {x=630.851, y=-229.172, z=22, rx=-180, rz=162.494, shoulder=lefty, elbow=epositive, wrist=wpositive, fatherId=fReference[0]}
  [2756] = {x=632.232, y=-228.737, z=22, rx=180, rz=162.332, shoulder=lefty, elbow=epositive, wrist=wpositive, fatherId=fReference[0]}
  [2757] = {x=633.612, y=-228.297, z=22, rx=-180, rz=162.171, shoulder=lefty, elbow=epositive, wrist=wpositive, fatherId=fReference[0]}
  [2758] = {x=634.991, y=-227.854, z=22, rx=180, rz=162.01, shoulder=lefty, elbow=epositive, wrist=wpositive, fatherId=fReference[0]}
  [2759] = {x=636.37, y=-227.406, z=22, rx=-180, rz=161.85, shoulder=lefty, elbow=epositive, wrist=wpositive, fatherId=fReference[0]}
  [2760] = {x=637.748, y=-226.954, z=22, rx=180, rz=161.69, shoulder=lefty, elbow=epositive, wrist=wpositive, fatherId=fReference[0]}
  [2761] = {x=639.125, y=-226.498, z=22, rx=180, rz=161.531, shoulder=lefty, elbow=epositive, wrist=wpositive, fatherId=fReference[0]}
  [2762] = {x=640.502, y=-226.038, z=22, rx=-180, rz=161.373, shoulder=lefty, elbow=epositive, wrist=wpositive, fatherId=fReference[0]}
  [2763] = {x=641.878, y=-225.575, z=22, rx=-180, rz=161.216, shoulder=lefty, elbow=epositive, wrist=wpositive, fatherId=fReference[0]}
  [2764] = {x=643.254, y=-225.107, z=22, rx=180, rz=161.059, shoulder=lefty, elbow=epositive, wrist=wpositive, fatherId=fReference[0]}
  [2765] = {x=644.628, y=-224.635, z=22, rx=-180, rz=160.903, shoulder=lefty, elbow=epositive, wrist=wpositive, fatherId=fReference[0]}
  [2766] = {x=646.002, y=-224.159, z=22, rx=180, rz=160.748, shoulder=lefty, elbow=epositive, wrist=wpositive, fatherId=fReference[0]}
  [2767] = {x=647.376, y=-223.68, z=22, rx=180, rz=160.593, shoulder=lefty, elbow=epositive, wrist=wpositive, fatherId=fReference[0]}
  [2768] = {x=648.748, y=-223.196, z=22, rx=-180, rz=160.439, shoulder=lefty, elbow=epositive, wrist=wpositive, fatherId=fReference[0]}
  [2769] = {x=650.12, y=-222.709, z=22, rx=-180, rz=160.286, shoulder=lefty, elbow=epositive, wrist=wpositive, fatherId=fReference[0]}
  [2770] = {x=651.491, y=-222.217, z=22, rx=180, rz=160.133, shoulder=lefty, elbow=epositive, wrist=wpositive, fatherId=fReference[0]}
  [2771] = {x=652.862, y=-221.722, z=22, rx=180, rz=159.981, shoulder=lefty, elbow=epositive, wrist=wpositive, fatherId=fReference[0]}
  [2772] = {x=654.232, y=-221.223, z=22, rx=-180, rz=159.83, shoulder=lefty, elbow=epositive, wrist=wpositive, fatherId=fReference[0]}
  [2773] = {x=655.601, y=-220.72, z=22, rx=180, rz=159.68, shoulder=lefty, elbow=epositive, wrist=wpositive, fatherId=fReference[0]}
  [2774] = {x=656.969, y=-220.213, z=22, rx=180, rz=159.53, shoulder=lefty, elbow=epositive, wrist=wpositive, fatherId=fReference[0]}
  [2775] = {x=658.337, y=-219.703, z=22, rx=180, rz=159.381, shoulder=lefty, elbow=epositive, wrist=wpositive, fatherId=fReference[0]}
  [2776] = {x=659.704, y=-219.189, z=22, rx=-180, rz=159.233, shoulder=lefty, elbow=epositive, wrist=wpositive, fatherId=fReference[0]}
  [2777] = {x=661.07, y=-218.67, z=22, rx=180, rz=159.086, shoulder=lefty, elbow=epositive, wrist=wpositive, fatherId=fReference[0]}
  [2778] = {x=662.436, y=-218.149, z=22, rx=180, rz=158.939, shoulder=lefty, elbow=epositive, wrist=wpositive, fatherId=fReference[0]}
  [2779] = {x=663.801, y=-217.623, z=22, rx=-180, rz=158.793, shoulder=lefty, elbow=epositive, wrist=wpositive, fatherId=fReference[0]}
  [2780] = {x=665.165, y=-217.094, z=22, rx=180, rz=158.647, shoulder=lefty, elbow=epositive, wrist=wpositive, fatherId=fReference[0]}
  [2781] = {x=666.528, y=-216.561, z=22, rx=-180, rz=158.503, shoulder=lefty, elbow=epositive, wrist=wpositive, fatherId=fReference[0]}
  [2782] = {x=667.891, y=-216.024, z=22, rx=180, rz=158.359, shoulder=lefty, elbow=epositive, wrist=wpositive, fatherId=fReference[0]}
  [2783] = {x=669.253, y=-215.484, z=22, rx=-180, rz=158.216, shoulder=lefty, elbow=epositive, wrist=wpositive, fatherId=fReference[0]}
  [2784] = {x=670.614, y=-214.94, z=22, rx=180, rz=158.073, shoulder=lefty, elbow=epositive, wrist=wpositive, fatherId=fReference[0]}
  [2785] = {x=671.974, y=-214.392, z=22, rx=180, rz=157.931, shoulder=lefty, elbow=epositive, wrist=wpositive, fatherId=fReference[0]}
  [2786] = {x=673.334, y=-213.841, z=22, rx=180, rz=157.79, shoulder=lefty, elbow=epositive, wrist=wpositive, fatherId=fReference[0]}
  [2787] = {x=674.693, y=-213.286, z=22, rx=180, rz=157.65, shoulder=lefty, elbow=epositive, wrist=wpositive, fatherId=fReference[0]}
  [2788] = {x=676.052, y=-212.727, z=22, rx=180, rz=157.51, shoulder=lefty, elbow=epositive, wrist=wpositive, fatherId=fReference[0]}
  [2789] = {x=677.409, y=-212.165, z=22, rx=180, rz=157.371, shoulder=lefty, elbow=epositive, wrist=wpositive, fatherId=fReference[0]}
  [2790] = {x=678.766, y=-211.6, z=22, rx=180, rz=157.233, shoulder=lefty, elbow=epositive, wrist=wpositive, fatherId=fReference[0]}
  [2791] = {x=680.122, y=-211.031, z=22, rx=-180, rz=157.096, shoulder=lefty, elbow=epositive, wrist=wpositive, fatherId=fReference[0]}
  [2792] = {x=681.477, y=-210.458, z=22, rx=180, rz=156.959, shoulder=lefty, elbow=epositive, wrist=wpositive, fatherId=fReference[0]}
  [2793] = {x=682.832, y=-209.882, z=22, rx=-180, rz=156.823, shoulder=lefty, elbow=epositive, wrist=wpositive, fatherId=fReference[0]}
  [2794] = {x=684.186, y=-209.302, z=22, rx=180, rz=156.688, shoulder=lefty, elbow=epositive, wrist=wpositive, fatherId=fReference[0]}
  [2795] = {x=685.539, y=-208.719, z=22, rx=-180, rz=156.553, shoulder=lefty, elbow=epositive, wrist=wpositive, fatherId=fReference[0]}
  [2796] = {x=686.891, y=-208.133, z=22, rx=-180, rz=156.42, shoulder=lefty, elbow=epositive, wrist=wpositive, fatherId=fReference[0]}
  [2797] = {x=688.243, y=-207.543, z=22, rx=180, rz=156.287, shoulder=lefty, elbow=epositive, wrist=wpositive, fatherId=fReference[0]}
  [2798] = {x=689.593, y=-206.949, z=22, rx=180, rz=156.154, shoulder=lefty, elbow=epositive, wrist=wpositive, fatherId=fReference[0]}
  [2799] = {x=690.943, y=-206.353, z=22, rx=180, rz=156.023, shoulder=lefty, elbow=epositive, wrist=wpositive, fatherId=fReference[0]}
  [2800] = {x=692.293, y=-205.753, z=22, rx=180, rz=155.892, shoulder=lefty, elbow=epositive, wrist=wpositive, fatherId=fReference[0]}
  [2801] = {x=693.641, y=-205.149, z=22, rx=-180, rz=155.762, shoulder=lefty, elbow=epositive, wrist=wpositive, fatherId=fReference[0]}
  [2802] = {x=694.989, y=-204.542, z=22, rx=-180, rz=155.632, shoulder=lefty, elbow=epositive, wrist=wpositive, fatherId=fReference[0]}
  [2803] = {x=696.336, y=-203.932, z=22, rx=180, rz=155.503, shoulder=lefty, elbow=epositive, wrist=wpositive, fatherId=fReference[0]}
  [2804] = {x=697.682, y=-203.319, z=22, rx=-180, rz=155.375, shoulder=lefty, elbow=epositive, wrist=wpositive, fatherId=fReference[0]}
  [2805] = {x=699.028, y=-202.702, z=22, rx=-180, rz=155.248, shoulder=lefty, elbow=epositive, wrist=wpositive, fatherId=fReference[0]}
  [2806] = {x=700.373, y=-202.082, z=22, rx=-180, rz=155.122, shoulder=lefty, elbow=epositive, wrist=wpositive, fatherId=fReference[0]}
  [2807] = {x=701.717, y=-201.459, z=22, rx=180, rz=154.996, shoulder=lefty, elbow=epositive, wrist=wpositive, fatherId=fReference[0]}
  [2808] = {x=703.06, y=-200.832, z=22, rx=-180, rz=154.871, shoulder=lefty, elbow=epositive, wrist=wpositive, fatherId=fReference[0]}
  [2809] = {x=704.403, y=-200.203, z=22, rx=-180, rz=154.746, shoulder=lefty, elbow=epositive, wrist=wpositive, fatherId=fReference[0]}
  [2810] = {x=705.744, y=-199.57, z=22, rx=-180, rz=154.622, shoulder=lefty, elbow=epositive, wrist=wpositive, fatherId=fReference[0]}
  [2811] = {x=707.085, y=-198.933, z=22, rx=-180, rz=154.499, shoulder=lefty, elbow=epositive, wrist=wpositive, fatherId=fReference[0]}
  [2812] = {x=708.426, y=-198.294, z=22, rx=180, rz=154.377, shoulder=lefty, elbow=epositive, wrist=wpositive, fatherId=fReference[0]}
  [2813] = {x=709.765, y=-197.652, z=22, rx=180, rz=154.256, shoulder=lefty, elbow=epositive, wrist=wpositive, fatherId=fReference[0]}
  [2814] = {x=711.104, y=-197.006, z=22, rx=-180, rz=154.135, shoulder=lefty, elbow=epositive, wrist=wpositive, fatherId=fReference[0]}
  [2815] = {x=712.442, y=-196.357, z=22, rx=-180, rz=154.015, shoulder=lefty, elbow=epositive, wrist=wpositive, fatherId=fReference[0]}
  [2816] = {x=713.779, y=-195.706, z=22, rx=180, rz=153.895, shoulder=lefty, elbow=epositive, wrist=wpositive, fatherId=fReference[0]}
  [2817] = {x=715.116, y=-195.051, z=22, rx=180, rz=153.776, shoulder=lefty, elbow=epositive, wrist=wpositive, fatherId=fReference[0]}
  [2818] = {x=716.452, y=-194.393, z=22, rx=180, rz=153.658, shoulder=lefty, elbow=epositive, wrist=wpositive, fatherId=fReference[0]}
  [2819] = {x=717.787, y=-193.732, z=22, rx=-180, rz=153.541, shoulder=lefty, elbow=epositive, wrist=wpositive, fatherId=fReference[0]}
  [2820] = {x=719.121, y=-193.067, z=22, rx=-180, rz=153.424, shoulder=lefty, elbow=epositive, wrist=wpositive, fatherId=fReference[0]}
  [2821] = {x=720.455, y=-192.4, z=22, rx=180, rz=153.309, shoulder=lefty, elbow=epositive, wrist=wpositive, fatherId=fReference[0]}
  [2822] = {x=721.788, y=-191.73, z=22, rx=-180, rz=153.193, shoulder=lefty, elbow=epositive, wrist=wpositive, fatherId=fReference[0]}
  [2823] = {x=723.12, y=-191.057, z=22, rx=-180, rz=153.079, shoulder=lefty, elbow=epositive, wrist=wpositive, fatherId=fReference[0]}
  [2824] = {x=724.451, y=-190.381, z=22, rx=-180, rz=152.965, shoulder=lefty, elbow=epositive, wrist=wpositive, fatherId=fReference[0]}
  [2825] = {x=725.782, y=-189.702, z=22, rx=-180, rz=152.852, shoulder=lefty, elbow=epositive, wrist=wpositive, fatherId=fReference[0]}
  [2826] = {x=727.112, y=-189.02, z=22, rx=-180, rz=152.739, shoulder=lefty, elbow=epositive, wrist=wpositive, fatherId=fReference[0]}
  [2827] = {x=728.441, y=-188.335, z=22, rx=-180, rz=152.628, shoulder=lefty, elbow=epositive, wrist=wpositive, fatherId=fReference[0]}
  [2828] = {x=729.77, y=-187.647, z=22, rx=180, rz=152.517, shoulder=lefty, elbow=epositive, wrist=wpositive, fatherId=fReference[0]}
  [2829] = {x=731.098, y=-186.957, z=22, rx=180, rz=152.406, shoulder=lefty, elbow=epositive, wrist=wpositive, fatherId=fReference[0]}
  [2830] = {x=732.425, y=-186.263, z=22, rx=-180, rz=152.297, shoulder=lefty, elbow=epositive, wrist=wpositive, fatherId=fReference[0]}
  [2831] = {x=733.751, y=-185.567, z=22, rx=180, rz=152.188, shoulder=lefty, elbow=epositive, wrist=wpositive, fatherId=fReference[0]}
  [2832] = {x=735.077, y=-184.867, z=22, rx=-180, rz=152.079, shoulder=lefty, elbow=epositive, wrist=wpositive, fatherId=fReference[0]}
  [2833] = {x=736.401, y=-184.165, z=22, rx=-180, rz=151.972, shoulder=lefty, elbow=epositive, wrist=wpositive, fatherId=fReference[0]}
  [2834] = {x=737.726, y=-183.46, z=22, rx=-180, rz=151.865, shoulder=lefty, elbow=epositive, wrist=wpositive, fatherId=fReference[0]}
  [2835] = {x=739.049, y=-182.753, z=22, rx=180, rz=151.759, shoulder=lefty, elbow=epositive, wrist=wpositive, fatherId=fReference[0]}
  [2836] = {x=740.372, y=-182.042, z=22, rx=-180, rz=151.653, shoulder=lefty, elbow=epositive, wrist=wpositive, fatherId=fReference[0]}
  [2837] = {x=741.694, y=-181.329, z=22, rx=-180, rz=151.548, shoulder=lefty, elbow=epositive, wrist=wpositive, fatherId=fReference[0]}
  [2838] = {x=743.015, y=-180.613, z=22, rx=180, rz=151.444, shoulder=lefty, elbow=epositive, wrist=wpositive, fatherId=fReference[0]}
  [2839] = {x=744.336, y=-179.894, z=22, rx=-180, rz=151.341, shoulder=lefty, elbow=epositive, wrist=wpositive, fatherId=fReference[0]}
  [2840] = {x=745.656, y=-179.173, z=22, rx=180, rz=151.238, shoulder=lefty, elbow=epositive, wrist=wpositive, fatherId=fReference[0]}
  [2841] = {x=746.975, y=-178.449, z=22, rx=-180, rz=151.136, shoulder=lefty, elbow=epositive, wrist=wpositive, fatherId=fReference[0]}
  [2842] = {x=748.293, y=-177.722, z=22, rx=180, rz=151.034, shoulder=lefty, elbow=epositive, wrist=wpositive, fatherId=fReference[0]}
  [2843] = {x=749.611, y=-176.993, z=22, rx=180, rz=150.933, shoulder=lefty, elbow=epositive, wrist=wpositive, fatherId=fReference[0]}
  [2844] = {x=750.928, y=-176.26, z=22, rx=-180, rz=150.833, shoulder=lefty, elbow=epositive, wrist=wpositive, fatherId=fReference[0]}
  [2845] = {x=752.244, y=-175.526, z=22, rx=180, rz=150.734, shoulder=lefty, elbow=epositive, wrist=wpositive, fatherId=fReference[0]}
  [2846] = {x=753.56, y=-174.788, z=22, rx=180, rz=150.635, shoulder=lefty, elbow=epositive, wrist=wpositive, fatherId=fReference[0]}
  [2847] = {x=754.875, y=-174.049, z=22, rx=180, rz=150.537, shoulder=lefty, elbow=epositive, wrist=wpositive, fatherId=fReference[0]}
  [2848] = {x=756.189, y=-173.306, z=22, rx=180, rz=150.439, shoulder=lefty, elbow=epositive, wrist=wpositive, fatherId=fReference[0]}
  [2849] = {x=757.503, y=-172.561, z=22, rx=180, rz=150.342, shoulder=lefty, elbow=epositive, wrist=wpositive, fatherId=fReference[0]}
  [2850] = {x=758.816, y=-171.814, z=22, rx=180, rz=150.246, shoulder=lefty, elbow=epositive, wrist=wpositive, fatherId=fReference[0]}
  [2851] = {x=760.128, y=-171.064, z=22, rx=180, rz=150.151, shoulder=lefty, elbow=epositive, wrist=wpositive, fatherId=fReference[0]}
  [2852] = {x=761.439, y=-170.311, z=22, rx=-180, rz=150.056, shoulder=lefty, elbow=epositive, wrist=wpositive, fatherId=fReference[0]}
  [2853] = {x=762.75, y=-169.556, z=22, rx=-180, rz=149.961, shoulder=lefty, elbow=epositive, wrist=wpositive, fatherId=fReference[0]}
  [2854] = {x=764.06, y=-168.798, z=22, rx=180, rz=149.868, shoulder=lefty, elbow=epositive, wrist=wpositive, fatherId=fReference[0]}
  [2855] = {x=765.369, y=-168.038, z=22, rx=180, rz=149.775, shoulder=lefty, elbow=epositive, wrist=wpositive, fatherId=fReference[0]}
  [2856] = {x=766.678, y=-167.276, z=22, rx=180, rz=149.683, shoulder=lefty, elbow=epositive, wrist=wpositive, fatherId=fReference[0]}
  [2857] = {x=767.986, y=-166.511, z=22, rx=180, rz=149.591, shoulder=lefty, elbow=epositive, wrist=wpositive, fatherId=fReference[0]}
  [2858] = {x=769.293, y=-165.744, z=22, rx=180, rz=149.5, shoulder=lefty, elbow=epositive, wrist=wpositive, fatherId=fReference[0]}
  [2859] = {x=770.6, y=-164.974, z=22, rx=180, rz=149.41, shoulder=lefty, elbow=epositive, wrist=wpositive, fatherId=fReference[0]}
  [2860] = {x=771.906, y=-164.202, z=22, rx=180, rz=149.32, shoulder=lefty, elbow=epositive, wrist=wpositive, fatherId=fReference[0]}
  [2861] = {x=773.211, y=-163.428, z=22, rx=180, rz=149.231, shoulder=lefty, elbow=epositive, wrist=wpositive, fatherId=fReference[0]}
  [2862] = {x=774.516, y=-162.651, z=22, rx=-180, rz=149.142, shoulder=lefty, elbow=epositive, wrist=wpositive, fatherId=fReference[0]}
  [2863] = {x=775.82, y=-161.872, z=22, rx=-180, rz=149.054, shoulder=lefty, elbow=epositive, wrist=wpositive, fatherId=fReference[0]}
  [2864] = {x=777.123, y=-161.091, z=22, rx=-180, rz=148.967, shoulder=lefty, elbow=epositive, wrist=wpositive, fatherId=fReference[0]}
  [2865] = {x=778.425, y=-160.307, z=22, rx=-180, rz=148.881, shoulder=lefty, elbow=epositive, wrist=wpositive, fatherId=fReference[0]}
  [2866] = {x=779.727, y=-159.521, z=22, rx=180, rz=148.795, shoulder=lefty, elbow=epositive, wrist=wpositive, fatherId=fReference[0]}
  [2867] = {x=781.028, y=-158.733, z=22, rx=-180, rz=148.709, shoulder=lefty, elbow=epositive, wrist=wpositive, fatherId=fReference[0]}
  [2868] = {x=782.329, y=-157.942, z=22, rx=180, rz=148.625, shoulder=lefty, elbow=epositive, wrist=wpositive, fatherId=fReference[0]}
  [2869] = {x=783.629, y=-157.15, z=22, rx=-180, rz=148.54, shoulder=lefty, elbow=epositive, wrist=wpositive, fatherId=fReference[0]}
  [2870] = {x=784.928, y=-156.355, z=22, rx=-180, rz=148.457, shoulder=lefty, elbow=epositive, wrist=wpositive, fatherId=fReference[0]}
  [2871] = {x=786.227, y=-155.558, z=22, rx=180, rz=148.374, shoulder=lefty, elbow=epositive, wrist=wpositive, fatherId=fReference[0]}
  [2872] = {x=787.524, y=-154.758, z=22, rx=180, rz=148.292, shoulder=lefty, elbow=epositive, wrist=wpositive, fatherId=fReference[0]}
  [2873] = {x=788.822, y=-153.957, z=22, rx=180, rz=148.21, shoulder=lefty, elbow=epositive, wrist=wpositive, fatherId=fReference[0]}
  [2874] = {x=790.118, y=-153.153, z=22, rx=180, rz=148.129, shoulder=lefty, elbow=epositive, wrist=wpositive, fatherId=fReference[0]}
  [2875] = {x=791.414, y=-152.348, z=22, rx=180, rz=148.049, shoulder=lefty, elbow=epositive, wrist=wpositive, fatherId=fReference[0]}
  [2876] = {x=792.709, y=-151.54, z=22, rx=180, rz=147.969, shoulder=lefty, elbow=epositive, wrist=wpositive, fatherId=fReference[0]}
  [2877] = {x=794.004, y=-150.73, z=22, rx=-180, rz=147.89, shoulder=lefty, elbow=epositive, wrist=wpositive, fatherId=fReference[0]}
  [2878] = {x=795.298, y=-149.918, z=22, rx=180, rz=147.811, shoulder=lefty, elbow=epositive, wrist=wpositive, fatherId=fReference[0]}
  [2879] = {x=796.591, y=-149.104, z=22, rx=180, rz=147.733, shoulder=lefty, elbow=epositive, wrist=wpositive, fatherId=fReference[0]}
  [2880] = {x=797.884, y=-148.288, z=22, rx=-180, rz=147.656, shoulder=lefty, elbow=epositive, wrist=wpositive, fatherId=fReference[0]}
  [2881] = {x=799.175, y=-147.47, z=22, rx=180, rz=147.579, shoulder=lefty, elbow=epositive, wrist=wpositive, fatherId=fReference[0]}
  [2882] = {x=800.467, y=-146.65, z=22, rx=-180, rz=147.503, shoulder=lefty, elbow=epositive, wrist=wpositive, fatherId=fReference[0]}
  [2883] = {x=801.757, y=-145.827, z=22, rx=180, rz=147.427, shoulder=lefty, elbow=epositive, wrist=wpositive, fatherId=fReference[0]}
  [2884] = {x=803.047, y=-145.003, z=22, rx=180, rz=147.352, shoulder=lefty, elbow=epositive, wrist=wpositive, fatherId=fReference[0]}
  [2885] = {x=804.337, y=-144.177, z=22, rx=180, rz=147.277, shoulder=lefty, elbow=epositive, wrist=wpositive, fatherId=fReference[0]}
  [2886] = {x=805.626, y=-143.349, z=22, rx=180, rz=147.204, shoulder=lefty, elbow=epositive, wrist=wpositive, fatherId=fReference[0]}
  [2887] = {x=806.914, y=-142.519, z=22, rx=-180, rz=147.13, shoulder=lefty, elbow=epositive, wrist=wpositive, fatherId=fReference[0]}
  [2888] = {x=808.201, y=-141.687, z=22, rx=-180, rz=147.058, shoulder=lefty, elbow=epositive, wrist=wpositive, fatherId=fReference[0]}
  [2889] = {x=809.488, y=-140.853, z=22, rx=180, rz=146.986, shoulder=lefty, elbow=epositive, wrist=wpositive, fatherId=fReference[0]}
  [2890] = {x=810.774, y=-140.017, z=22, rx=-180, rz=146.914, shoulder=lefty, elbow=epositive, wrist=wpositive, fatherId=fReference[0]}
  [2891] = {x=812.06, y=-139.18, z=22, rx=-180, rz=146.843, shoulder=lefty, elbow=epositive, wrist=wpositive, fatherId=fReference[0]}
  [2892] = {x=813.345, y=-138.34, z=22, rx=-180, rz=146.773, shoulder=lefty, elbow=epositive, wrist=wpositive, fatherId=fReference[0]}
  [2893] = {x=814.629, y=-137.499, z=22, rx=-180, rz=146.703, shoulder=lefty, elbow=epositive, wrist=wpositive, fatherId=fReference[0]}
  [2894] = {x=815.913, y=-136.656, z=22, rx=180, rz=146.634, shoulder=lefty, elbow=epositive, wrist=wpositive, fatherId=fReference[0]}
  [2895] = {x=817.196, y=-135.811, z=22, rx=180, rz=146.565, shoulder=lefty, elbow=epositive, wrist=wpositive, fatherId=fReference[0]}
  [2896] = {x=818.479, y=-134.964, z=22, rx=-180, rz=146.497, shoulder=lefty, elbow=epositive, wrist=wpositive, fatherId=fReference[0]}
  [2897] = {x=819.761, y=-134.115, z=22, rx=180, rz=146.429, shoulder=lefty, elbow=epositive, wrist=wpositive, fatherId=fReference[0]}
  [2898] = {x=821.042, y=-133.265, z=22, rx=-180, rz=146.362, shoulder=lefty, elbow=epositive, wrist=wpositive, fatherId=fReference[0]}
  [2899] = {x=822.323, y=-132.413, z=22, rx=-180, rz=146.296, shoulder=lefty, elbow=epositive, wrist=wpositive, fatherId=fReference[0]}
  [2900] = {x=823.603, y=-131.559, z=22, rx=180, rz=146.23, shoulder=lefty, elbow=epositive, wrist=wpositive, fatherId=fReference[0]}
  [2901] = {x=824.882, y=-130.703, z=22, rx=-180, rz=146.165, shoulder=lefty, elbow=epositive, wrist=wpositive, fatherId=fReference[0]}
  [2902] = {x=826.161, y=-129.846, z=22, rx=180, rz=146.1, shoulder=lefty, elbow=epositive, wrist=wpositive, fatherId=fReference[0]}
  [2903] = {x=827.44, y=-128.987, z=22, rx=180, rz=146.036, shoulder=lefty, elbow=epositive, wrist=wpositive, fatherId=fReference[0]}
  [2904] = {x=828.717, y=-128.127, z=22, rx=-180, rz=145.972, shoulder=lefty, elbow=epositive, wrist=wpositive, fatherId=fReference[0]}
  [2905] = {x=829.994, y=-127.264, z=22, rx=180, rz=145.909, shoulder=lefty, elbow=epositive, wrist=wpositive, fatherId=fReference[0]}
  [2906] = {x=831.271, y=-126.4, z=22, rx=180, rz=145.847, shoulder=lefty, elbow=epositive, wrist=wpositive, fatherId=fReference[0]}
  [2907] = {x=832.547, y=-125.535, z=22, rx=180, rz=145.785, shoulder=lefty, elbow=epositive, wrist=wpositive, fatherId=fReference[0]}
  [2908] = {x=833.822, y=-124.667, z=22, rx=-180, rz=145.723, shoulder=lefty, elbow=epositive, wrist=wpositive, fatherId=fReference[0]}
  [2909] = {x=835.097, y=-123.798, z=22, rx=180, rz=145.662, shoulder=lefty, elbow=epositive, wrist=wpositive, fatherId=fReference[0]}
  [2910] = {x=836.372, y=-122.928, z=22, rx=-180, rz=145.602, shoulder=lefty, elbow=epositive, wrist=wpositive, fatherId=fReference[0]}
  [2911] = {x=837.645, y=-122.056, z=22, rx=180, rz=145.542, shoulder=lefty, elbow=epositive, wrist=wpositive, fatherId=fReference[0]}
  [2912] = {x=838.918, y=-121.182, z=22, rx=-180, rz=145.483, shoulder=lefty, elbow=epositive, wrist=wpositive, fatherId=fReference[0]}
  [2913] = {x=840.191, y=-120.307, z=22, rx=180, rz=145.424, shoulder=lefty, elbow=epositive, wrist=wpositive, fatherId=fReference[0]}
  [2914] = {x=841.463, y=-119.43, z=22, rx=180, rz=145.366, shoulder=lefty, elbow=epositive, wrist=wpositive, fatherId=fReference[0]}
  [2915] = {x=842.734, y=-118.552, z=22, rx=-180, rz=145.308, shoulder=lefty, elbow=epositive, wrist=wpositive, fatherId=fReference[0]}
  [2916] = {x=844.005, y=-117.672, z=22, rx=180, rz=145.251, shoulder=lefty, elbow=epositive, wrist=wpositive, fatherId=fReference[0]}
  [2917] = {x=845.276, y=-116.791, z=22, rx=180, rz=145.195, shoulder=lefty, elbow=epositive, wrist=wpositive, fatherId=fReference[0]}
  [2918] = {x=846.545, y=-115.908, z=22, rx=180, rz=145.139, shoulder=lefty, elbow=epositive, wrist=wpositive, fatherId=fReference[0]}
  [2919] = {x=847.815, y=-115.024, z=22, rx=180, rz=145.083, shoulder=lefty, elbow=epositive, wrist=wpositive, fatherId=fReference[0]}
  [2920] = {x=849.084, y=-114.139, z=22, rx=-180, rz=145.028, shoulder=lefty, elbow=epositive, wrist=wpositive, fatherId=fReference[0]}
  [2921] = {x=850.352, y=-113.251, z=22, rx=-180, rz=144.974, shoulder=lefty, elbow=epositive, wrist=wpositive, fatherId=fReference[0]}
  [2922] = {x=851.619, y=-112.363, z=22, rx=180, rz=144.92, shoulder=lefty, elbow=epositive, wrist=wpositive, fatherId=fReference[0]}
  [2923] = {x=852.887, y=-111.473, z=22, rx=-180, rz=144.866, shoulder=lefty, elbow=epositive, wrist=wpositive, fatherId=fReference[0]}
  [2924] = {x=854.153, y=-110.582, z=22, rx=180, rz=144.813, shoulder=lefty, elbow=epositive, wrist=wpositive, fatherId=fReference[0]}
  [2925] = {x=855.419, y=-109.689, z=22, rx=180, rz=144.761, shoulder=lefty, elbow=epositive, wrist=wpositive, fatherId=fReference[0]}
  [2926] = {x=856.685, y=-108.795, z=22, rx=180, rz=144.709, shoulder=lefty, elbow=epositive, wrist=wpositive, fatherId=fReference[0]}
  [2927] = {x=857.95, y=-107.899, z=22, rx=-180, rz=144.657, shoulder=lefty, elbow=epositive, wrist=wpositive, fatherId=fReference[0]}
  [2928] = {x=859.215, y=-107.003, z=22, rx=180, rz=144.607, shoulder=lefty, elbow=epositive, wrist=wpositive, fatherId=fReference[0]}
  [2929] = {x=860.479, y=-106.104, z=22, rx=180, rz=144.556, shoulder=lefty, elbow=epositive, wrist=wpositive, fatherId=fReference[0]}
  [2930] = {x=861.742, y=-105.205, z=22, rx=180, rz=144.506, shoulder=lefty, elbow=epositive, wrist=wpositive, fatherId=fReference[0]}
  [2931] = {x=863.006, y=-104.304, z=22, rx=180, rz=144.457, shoulder=lefty, elbow=epositive, wrist=wpositive, fatherId=fReference[0]}
  [2932] = {x=864.268, y=-103.402, z=22, rx=180, rz=144.408, shoulder=lefty, elbow=epositive, wrist=wpositive, fatherId=fReference[0]}
  [2933] = {x=865.53, y=-102.499, z=22, rx=180, rz=144.36, shoulder=lefty, elbow=epositive, wrist=wpositive, fatherId=fReference[0]}
  [2934] = {x=866.792, y=-101.594, z=22, rx=-180, rz=144.312, shoulder=lefty, elbow=epositive, wrist=wpositive, fatherId=fReference[0]}
  [2935] = {x=868.053, y=-100.688, z=22, rx=-180, rz=144.265, shoulder=lefty, elbow=epositive, wrist=wpositive, fatherId=fReference[0]}
  [2936] = {x=869.314, y=-99.781, z=22, rx=180, rz=144.218, shoulder=lefty, elbow=epositive, wrist=wpositive, fatherId=fReference[0]}
  [2937] = {x=870.574, y=-98.873, z=22, rx=180, rz=144.172, shoulder=lefty, elbow=epositive, wrist=wpositive, fatherId=fReference[0]}
  [2938] = {x=871.834, y=-97.963, z=22, rx=180, rz=144.126, shoulder=lefty, elbow=epositive, wrist=wpositive, fatherId=fReference[0]}
  [2939] = {x=873.094, y=-97.052, z=22, rx=180, rz=144.08, shoulder=lefty, elbow=epositive, wrist=wpositive, fatherId=fReference[0]}
  [2940] = {x=874.353, y=-96.14, z=22, rx=180, rz=144.036, shoulder=lefty, elbow=epositive, wrist=wpositive, fatherId=fReference[0]}
  [2941] = {x=875.611, y=-95.227, z=22, rx=-180, rz=143.991, shoulder=lefty, elbow=epositive, wrist=wpositive, fatherId=fReference[0]}
  [2942] = {x=876.869, y=-94.313, z=22, rx=180, rz=143.947, shoulder=lefty, elbow=epositive, wrist=wpositive, fatherId=fReference[0]}
  [2943] = {x=878.127, y=-93.397, z=22, rx=-180, rz=143.904, shoulder=lefty, elbow=epositive, wrist=wpositive, fatherId=fReference[0]}
  [2944] = {x=879.384, y=-92.481, z=22, rx=-180, rz=143.861, shoulder=lefty, elbow=epositive, wrist=wpositive, fatherId=fReference[0]}
  [2945] = {x=880.641, y=-91.563, z=22, rx=180, rz=143.819, shoulder=lefty, elbow=epositive, wrist=wpositive, fatherId=fReference[0]}
  [2946] = {x=881.897, y=-90.644, z=22, rx=180, rz=143.777, shoulder=lefty, elbow=epositive, wrist=wpositive, fatherId=fReference[0]}
  [2947] = {x=883.153, y=-89.724, z=22, rx=180, rz=143.735, shoulder=lefty, elbow=epositive, wrist=wpositive, fatherId=fReference[0]}
  [2948] = {x=884.409, y=-88.803, z=22, rx=180, rz=143.694, shoulder=lefty, elbow=epositive, wrist=wpositive, fatherId=fReference[0]}
  [2949] = {x=885.664, y=-87.881, z=22, rx=180, rz=143.654, shoulder=lefty, elbow=epositive, wrist=wpositive, fatherId=fReference[0]}
  [2950] = {x=886.919, y=-86.957, z=22, rx=-180, rz=143.614, shoulder=lefty, elbow=epositive, wrist=wpositive, fatherId=fReference[0]}
  [2951] = {x=888.173, y=-86.033, z=22, rx=180, rz=143.574, shoulder=lefty, elbow=epositive, wrist=wpositive, fatherId=fReference[0]}
  [2952] = {x=889.427, y=-85.108, z=22, rx=180, rz=143.535, shoulder=lefty, elbow=epositive, wrist=wpositive, fatherId=fReference[0]}
  [2953] = {x=890.681, y=-84.181, z=22, rx=180, rz=143.497, shoulder=lefty, elbow=epositive, wrist=wpositive, fatherId=fReference[0]}
  [2954] = {x=891.934, y=-83.254, z=22, rx=-180, rz=143.459, shoulder=lefty, elbow=epositive, wrist=wpositive, fatherId=fReference[0]}
  [2955] = {x=893.187, y=-82.325, z=22, rx=-180, rz=143.421, shoulder=lefty, elbow=epositive, wrist=wpositive, fatherId=fReference[0]}
  [2956] = {x=894.439, y=-81.396, z=22, rx=180, rz=143.384, shoulder=lefty, elbow=epositive, wrist=wpositive, fatherId=fReference[0]}
  [2957] = {x=895.691, y=-80.465, z=22, rx=180, rz=143.347, shoulder=lefty, elbow=epositive, wrist=wpositive, fatherId=fReference[0]}
  [2958] = {x=896.943, y=-79.534, z=22, rx=180, rz=143.311, shoulder=lefty, elbow=epositive, wrist=wpositive, fatherId=fReference[0]}
  [2959] = {x=898.195, y=-78.602, z=22, rx=180, rz=143.275, shoulder=lefty, elbow=epositive, wrist=wpositive, fatherId=fReference[0]}
  [2960] = {x=899.446, y=-77.668, z=22, rx=180, rz=143.24, shoulder=lefty, elbow=epositive, wrist=wpositive, fatherId=fReference[0]}
  [2961] = {x=900.696, y=-76.734, z=22, rx=-180, rz=143.205, shoulder=lefty, elbow=epositive, wrist=wpositive, fatherId=fReference[0]}
  [2962] = {x=901.947, y=-75.799, z=22, rx=-180, rz=143.171, shoulder=lefty, elbow=epositive, wrist=wpositive, fatherId=fReference[0]}
  [2963] = {x=903.197, y=-74.862, z=22, rx=-180, rz=143.137, shoulder=lefty, elbow=epositive, wrist=wpositive, fatherId=fReference[0]}
  [2964] = {x=904.447, y=-73.925, z=22, rx=-180, rz=143.103, shoulder=lefty, elbow=epositive, wrist=wpositive, fatherId=fReference[0]}
  [2965] = {x=905.696, y=-72.987, z=22, rx=180, rz=143.07, shoulder=lefty, elbow=epositive, wrist=wpositive, fatherId=fReference[0]}
  [2966] = {x=906.945, y=-72.049, z=22, rx=180, rz=143.038, shoulder=lefty, elbow=epositive, wrist=wpositive, fatherId=fReference[0]}
  [2967] = {x=908.194, y=-71.109, z=22, rx=180, rz=143.006, shoulder=lefty, elbow=epositive, wrist=wpositive, fatherId=fReference[0]}
  [2968] = {x=909.442, y=-70.168, z=22, rx=180, rz=142.974, shoulder=lefty, elbow=epositive, wrist=wpositive, fatherId=fReference[0]}
  [2969] = {x=910.69, y=-69.227, z=22, rx=-180, rz=142.943, shoulder=lefty, elbow=epositive, wrist=wpositive, fatherId=fReference[0]}
  [2970] = {x=911.938, y=-68.285, z=22, rx=180, rz=142.912, shoulder=lefty, elbow=epositive, wrist=wpositive, fatherId=fReference[0]}
  [2971] = {x=913.185, y=-67.342, z=22, rx=-180, rz=142.882, shoulder=lefty, elbow=epositive, wrist=wpositive, fatherId=fReference[0]}
  [2972] = {x=914.433, y=-66.398, z=22, rx=180, rz=142.853, shoulder=lefty, elbow=epositive, wrist=wpositive, fatherId=fReference[0]}
  [2973] = {x=915.68, y=-65.453, z=22, rx=180, rz=142.823, shoulder=lefty, elbow=epositive, wrist=wpositive, fatherId=fReference[0]}
  [2974] = {x=916.926, y=-64.508, z=22, rx=-180, rz=142.794, shoulder=lefty, elbow=epositive, wrist=wpositive, fatherId=fReference[0]}
  [2975] = {x=918.172, y=-63.562, z=22, rx=-180, rz=142.766, shoulder=lefty, elbow=epositive, wrist=wpositive, fatherId=fReference[0]}
  [2976] = {x=919.418, y=-62.615, z=22, rx=-180, rz=142.738, shoulder=lefty, elbow=epositive, wrist=wpositive, fatherId=fReference[0]}
  [2977] = {x=920.664, y=-61.667, z=22, rx=-180, rz=142.71, shoulder=lefty, elbow=epositive, wrist=wpositive, fatherId=fReference[0]}
  [2978] = {x=921.91, y=-60.719, z=22, rx=-180, rz=142.683, shoulder=lefty, elbow=epositive, wrist=wpositive, fatherId=fReference[0]}
  [2979] = {x=923.155, y=-59.769, z=22, rx=180, rz=142.657, shoulder=lefty, elbow=epositive, wrist=wpositive, fatherId=fReference[0]}
  [2980] = {x=924.4, y=-58.82, z=22, rx=180, rz=142.631, shoulder=lefty, elbow=epositive, wrist=wpositive, fatherId=fReference[0]}
  [2981] = {x=925.644, y=-57.869, z=22, rx=-180, rz=142.605, shoulder=lefty, elbow=epositive, wrist=wpositive, fatherId=fReference[0]}
  [2982] = {x=926.889, y=-56.918, z=22, rx=-180, rz=142.58, shoulder=lefty, elbow=epositive, wrist=wpositive, fatherId=fReference[0]}
  [2983] = {x=928.133, y=-55.966, z=22, rx=180, rz=142.555, shoulder=lefty, elbow=epositive, wrist=wpositive, fatherId=fReference[0]}
  [2984] = {x=929.377, y=-55.013, z=22, rx=180, rz=142.53, shoulder=lefty, elbow=epositive, wrist=wpositive, fatherId=fReference[0]}
  [2985] = {x=930.621, y=-54.06, z=22, rx=180, rz=142.507, shoulder=lefty, elbow=epositive, wrist=wpositive, fatherId=fReference[0]}
  [2986] = {x=931.864, y=-53.106, z=22, rx=180, rz=142.483, shoulder=lefty, elbow=epositive, wrist=wpositive, fatherId=fReference[0]}
  [2987] = {x=933.107, y=-52.152, z=22, rx=180, rz=142.46, shoulder=lefty, elbow=epositive, wrist=wpositive, fatherId=fReference[0]}
  [2988] = {x=934.35, y=-51.197, z=22, rx=180, rz=142.437, shoulder=lefty, elbow=epositive, wrist=wpositive, fatherId=fReference[0]}
  [2989] = {x=935.593, y=-50.241, z=22, rx=180, rz=142.415, shoulder=lefty, elbow=epositive, wrist=wpositive, fatherId=fReference[0]}
  [2990] = {x=936.835, y=-49.284, z=22, rx=180, rz=142.393, shoulder=lefty, elbow=epositive, wrist=wpositive, fatherId=fReference[0]}
  [2991] = {x=938.078, y=-48.328, z=22, rx=180, rz=142.372, shoulder=lefty, elbow=epositive, wrist=wpositive, fatherId=fReference[0]}
  [2992] = {x=939.32, y=-47.37, z=22, rx=-180, rz=142.351, shoulder=lefty, elbow=epositive, wrist=wpositive, fatherId=fReference[0]}
  [2993] = {x=940.561, y=-46.412, z=22, rx=180, rz=142.331, shoulder=lefty, elbow=epositive, wrist=wpositive, fatherId=fReference[0]}
  [2994] = {x=941.803, y=-45.454, z=22, rx=180, rz=142.311, shoulder=lefty, elbow=epositive, wrist=wpositive, fatherId=fReference[0]}
  [2995] = {x=943.044, y=-44.494, z=22, rx=-180, rz=142.291, shoulder=lefty, elbow=epositive, wrist=wpositive, fatherId=fReference[0]}
  [2996] = {x=944.286, y=-43.535, z=22, rx=-180, rz=142.272, shoulder=lefty, elbow=epositive, wrist=wpositive, fatherId=fReference[0]}
  [2997] = {x=945.527, y=-42.575, z=22, rx=180, rz=142.254, shoulder=lefty, elbow=epositive, wrist=wpositive, fatherId=fReference[0]}
  [2998] = {x=946.768, y=-41.614, z=22, rx=-180, rz=142.235, shoulder=lefty, elbow=epositive, wrist=wpositive, fatherId=fReference[0]}
  [2999] = {x=948.008, y=-40.653, z=22, rx=-180, rz=142.217, shoulder=lefty, elbow=epositive, wrist=wpositive, fatherId=fReference[0]}
  [3000] = {x=949.249, y=-39.691, z=22, rx=180, rz=142.2, shoulder=lefty, elbow=epositive, wrist=wpositive, fatherId=fReference[0]}
  [3001] = {x=950.489, y=-38.729, z=22, rx=180, rz=142.183, shoulder=lefty, elbow=epositive, wrist=wpositive, fatherId=fReference[0]}
  [3002] = {x=951.729, y=-37.767, z=22, rx=-180, rz=142.167, shoulder=lefty, elbow=epositive, wrist=wpositive, fatherId=fReference[0]}
  [3003] = {x=952.969, y=-36.804, z=22, rx=180, rz=142.151, shoulder=lefty, elbow=epositive, wrist=wpositive, fatherId=fReference[0]}
  [3004] = {x=954.209, y=-35.841, z=22, rx=180, rz=142.135, shoulder=lefty, elbow=epositive, wrist=wpositive, fatherId=fReference[0]}
  [3005] = {x=955.448, y=-34.877, z=22, rx=180, rz=142.12, shoulder=lefty, elbow=epositive, wrist=wpositive, fatherId=fReference[0]}
  [3006] = {x=956.688, y=-33.913, z=22, rx=-180, rz=142.105, shoulder=lefty, elbow=epositive, wrist=wpositive, fatherId=fReference[0]}
  [3007] = {x=957.927, y=-32.948, z=22, rx=180, rz=142.09, shoulder=lefty, elbow=epositive, wrist=wpositive, fatherId=fReference[0]}
  [3008] = {x=959.166, y=-31.983, z=22, rx=-180, rz=142.076, shoulder=lefty, elbow=epositive, wrist=wpositive, fatherId=fReference[0]}
  [3009] = {x=960.405, y=-31.018, z=22, rx=180, rz=142.063, shoulder=lefty, elbow=epositive, wrist=wpositive, fatherId=fReference[0]}
  [3010] = {x=961.644, y=-30.052, z=22, rx=180, rz=142.05, shoulder=lefty, elbow=epositive, wrist=wpositive, fatherId=fReference[0]}
  [3011] = {x=962.882, y=-29.086, z=22, rx=180, rz=142.037, shoulder=lefty, elbow=epositive, wrist=wpositive, fatherId=fReference[0]}
  [3012] = {x=964.121, y=-28.12, z=22, rx=-180, rz=142.025, shoulder=lefty, elbow=epositive, wrist=wpositive, fatherId=fReference[0]}
  [3013] = {x=965.359, y=-27.153, z=22, rx=180, rz=142.013, shoulder=lefty, elbow=epositive, wrist=wpositive, fatherId=fReference[0]}
  [3014] = {x=966.598, y=-26.186, z=22, rx=-180, rz=142.002, shoulder=lefty, elbow=epositive, wrist=wpositive, fatherId=fReference[0]}
  [3015] = {x=967.836, y=-25.219, z=22, rx=-180, rz=141.991, shoulder=lefty, elbow=epositive, wrist=wpositive, fatherId=fReference[0]}
  [3016] = {x=969.074, y=-24.251, z=22, rx=-180, rz=141.98, shoulder=lefty, elbow=epositive, wrist=wpositive, fatherId=fReference[0]}
  [3017] = {x=970.312, y=-23.283, z=22, rx=-180, rz=141.97, shoulder=lefty, elbow=epositive, wrist=wpositive, fatherId=fReference[0]}
